// TIA Portal V20 program export: 1 tag tables, 32 data types, 19 data blocks, 60 code blocks (in call order from the OBs), 16 instance data blocks

VAR_GLOBAL   // PLC tag table "IMC88"
   IMC88Sensor_1 AT %I727.0 : Bool;   // High = Sensor active (input type and polarity can be configured)
   IMC88Sensor_2 AT %I727.1 : Bool;   // High = Sensor active (input type and polarity can be configured)
   IMC88Sensor_3 AT %I727.2 : Bool;   // High = Sensor active (input type and polarity can be configured)
   IMC88Sensor_4 AT %I727.3 : Bool;   // High = Sensor active (input type and polarity can be configured)
   IMC88Sensor_5 AT %I727.4 : Bool;
   IMC88Sensor_6 AT %I727.5 : Bool;
   IMC88Sensor_7 AT %I727.6 : Bool;
   IMC88Sensor_8 AT %I727.7 : Bool;
   IMC88IO1 AT %I728.0 : Bool;   // Digital I/O PLC Input PLC Output
   IMC88IO2 AT %I728.1 : Bool;   // Digital I/O PLC Input PLC Output
   IMC88IO3 AT %I728.2 : Bool;   // Digital I/O PLC Input PLC Output
   IMC88IO4 AT %I728.3 : Bool;   // Digital I/O PLC Input PLC Output
   IMC88IO5 AT %I728.4 : Bool;
   IMC88IO6 AT %I728.5 : Bool;
   IMC88IO7 AT %I728.6 : Bool;
   IMC88IO8 AT %I728.7 : Bool;
   "IMC88MotorStateErrorRD -G1.7.4" AT %I729.0 : Bool;   // High = Motor Error; Low = Motor OK
   "IMC88MotorStateErrorRD -G1.7.3" AT %I729.1 : Bool;   // High = Motor Error; Low = Motor OK
   "IMC88MotorStateErrorRD -G1.7.2" AT %I729.2 : Bool;   // High = Motor Error; Low = Motor OK
   "IMC88MotorStateErrorRD -4" AT %I729.3 : Bool;   // High = Motor Error; Low = Motor OK
   "IMC88MotorStateSpeedRD -G1.7.4" AT %IB730 : SInt;   // Speed 0–100 ( 0 = Stop, 100 = max speed), negative sign reverses the turning direction
   "IMC88MotorStateSpeedRD -G1.7.3" AT %IB731 : SInt;   // Speed 0–100 ( 0 = Stop, 100 = max speed), negative sign reverses the turning direction
   "IMC88MotorStateSpeedRD -G1.7.2" AT %IB732 : SInt;   // Speed 0–100 ( 0 = Stop, 100 = max speed), negative sign reverses the turning direction
   "IMC88MotorStateSpeedRD -4" AT %IB733 : SInt;   // Speed 0–100 ( 0 = Stop, 100 = max speed), negative sign reverses the turning direction
   "IMC88MotorCurrentRD -G1.7.4" AT %IW735 : Int;   // Average current in mA
   "IMC88MotorCurrentRD -G1.7.3" AT %IW737 : Int;   // Average current in mA
   "IMC88MotorCurrentRD -G1.7.2" AT %IW739 : Int;   // Average current in mA
   "IMC88MotorCurrentRD -4" AT %IW741 : Int;   // Average current in mA
   "IMC88Voltage(MotorPower)" AT %IW743 : Int;   // Voltage „Motor Power“ in mV
   "IMC88Voltage(Sensors)" AT %IW745 : Int;   // Voltage „Power Logic + Sensors“ in mV
   IMC88Temperature AT %IW747 : Int;   // Temperature in 0,1 C
   IMC88SystemUpTime AT %ID749 : DInt;   // Operating time in seconds since the last start/restart
   "IMC88DigitalOutputRD -G1.7.4" AT %Q535.0 : Bool;
   "IMC88DigitalOutputRD -G1.7.3" AT %Q535.1 : Bool;
   "IMC88DigitalOutputRD -G1.7.2" AT %Q535.2 : Bool;
   "IMC88DigitalOutputRD -4" AT %Q535.3 : Bool;
   "IMC88MotorTargetSpeedRD -G1.7.4" AT %QB536 : SInt;   // Speed 0–100 ( 0 = Stop, 100 = max speed), negative sign reverses the turning direction
   "IMC88MotorTargetSpeedRD -G1.7.3" AT %QB537 : SInt;   // Speed 0–100 ( 0 = Stop, 100 = max speed), negative sign reverses the turning direction
   "IMC88MotorTargetSpeedRD -G1.7.2" AT %QB538 : SInt;   // Speed 0–100 ( 0 = Stop, 100 = max speed), negative sign reverses the turning direction
   "IMC88MotorTargetSpeedRD -4" AT %QB539 : SInt;   // Speed 0–100 ( 0 = Stop, 100 = max speed), negative sign reverses the turning direction
END_VAR

TYPE "BarCode"
// stored: Access Published, Namespace Global
   STRUCT
      "Result Data" : Array[0..63] of Byte;
   END_STRUCT;
END_TYPE

TYPE "ConveyorParameters"
// stored: Access Published, Namespace Global
   STRUCT
      StartUpTime : Time := T#0S;
      SensorFilterTime : Array[1..2] of Time;
      SensorBlockageTime : Time := T#5S;
      EnergySaveTime : Time := T#3s;
      ConvOccTime : Time := T#1000ms;
      "IMC-SpeedSetPoint" : SInt := 100;
   END_STRUCT;
   // SensorFilterTime[1..2] := T#10ms;
END_TYPE

TYPE "ConveyorParameters_TransferUnit"
// stored: Access Published, Namespace Global
   STRUCT
      StartUpTime : Time := T#0S;
      SensorFilterTime : Array[1..2] of Time;
      FrontSensorFilterTime : Array[1..2] of Time;
      "Left/RightSensorFilterTime" : Array[1..2] of Time;
      EndsensorFilterTime : Array[1..2] of Time;
      SensorBlockageTime : Time := T#5S;
      EnergySaveTime : Time := T#3s;
      ConvOccTime : Time := T#1000ms;
   END_STRUCT;
   // SensorFilterTime[1..2] := T#10ms;
   // FrontSensorFilterTime[1..2] := T#10ms;
   // "Left/RightSensorFilterTime"[1..2] := T#10ms;
END_TYPE

TYPE "ConveyorStatus"
// stored: Access Published, Namespace Global
   STRUCT
      Blockage : Bool;
      xReserved_2 : Bool;
      xReserved_3 : Bool;
      xReserved_4 : Bool;
      xReserved_5 : Bool;
      xReserved_6 : Bool;
      xReserved_7 : Bool;
      xReserved_8 : Bool;
      ON : Bool;
      ReadytoRun : Bool;
      Occupied : Bool;
      Running : Bool;
      Fault : Bool;
      Estop : Bool;
      Manual : Bool;
      Stop : Bool;
   END_STRUCT;
END_TYPE

TYPE "EsopZone"
// stored: Access Published, Namespace Global
   STRUCT
      "1" : Bool;
      "2" : Bool;
   END_STRUCT;
END_TYPE

TYPE "Fault"
// stored: Access Published, Namespace Global
   STRUCT
      Motor_Error : Bool;
      Sensor_Blockage : Bool;
   END_STRUCT;
END_TYPE

TYPE "GetDiag"
// stored: Access Published, Namespace Global
   STRUCT
      DiagMode : UInt := 1;
      CommID : HW_ANY;
      ReturnValue : Int;
      CountDiagDetail : UInt;
      MyDiag : DIS;
   END_STRUCT;
END_TYPE

TYPE "ItemDir"
// stored: Access Published, Namespace Global
   STRUCT
      Straight : Bool;
      toRight : Bool;
      toLeft : Bool;
   END_STRUCT;
END_TYPE

TYPE "MABS_Parameters"
// stored: Access Published, Namespace Global
   STRUCT
      StartUpTime : Time := T#5S;
      CrossSensorFilterTime : Array[1..2] of Time;
      SensorBlockageTime : Time := T#5S;
      EnergySaveTime : Time := T#4s;
   END_STRUCT;
END_TYPE

TYPE "ManualInputs"
// stored: Access Published, Namespace Global
   STRUCT
      ManualEnable : Bool;
      Run : Struct
         Forward : Bool;
         Reverse : Bool;
      END_STRUCT;
   END_STRUCT;
END_TYPE

TYPE "S300ForceMode"
// stored: Access Published, Namespace Global
   STRUCT
      BeltDir : Bool;
      RollerDir : Bool;
   END_STRUCT;
END_TYPE

TYPE "S300Manual"
// stored: Namespace Global
   STRUCT
      GoUp : Bool;
      GoStraight : Bool;
      GoLeft : Bool;
      GoRight : Bool;
   END_STRUCT;
END_TYPE

TYPE "SystemSSR"
// stored: Access Published, Namespace Global
   STRUCT
      StartSystem : Bool;   // Start the system
      StopSystem : Bool;   // Stop the system
      ResetSystem : Bool;   // Reset the system
   END_STRUCT;
END_TYPE

TYPE "TrackingData"
// stored: Access Published, Namespace Global
   STRUCT
      Barcode : String;
      ResponseCode : UInt;
      HeightLimit : Bool;
      ActualWeight : Struct
         inRealValue : Real;
         inStringFormat : String;
      END_STRUCT;
      EXIT_1_ : Array[1..1] of Bool;
      EXIT_2_ : Array[1..6] of Bool;
      ToteDir : "Global.ItemDir";
   END_STRUCT;
END_TYPE

TYPE "IB_P01_02_03_in_64bytes_struct"
// stored: Access Published, Namespace Global
   STRUCT
      Reserved : Byte;
      Sens_A : Bool;
      Sens_B : Bool;
      Sens_A_alrm : Bool;
      Sens_B_alrm : Bool;
      Motor_state_A : Bool;
      Motor_state_B : Bool;
      Reserved_1 : Bool;
      Reserved_2 : Bool;
      Fuse_err_A : Bool;
      Back_EMF_err_A : Bool;
      Thermal_err_mot_A : Bool;
      Thermal_err_ctrl_A : Bool;
      Lock_err_A : Bool;
      Unconnected_err_A : Bool;
      Reserved_3 : Bool;
      Reserved_4 : Bool;
      Fuse_err_B : Bool;
      Back_EMF_err_B : Bool;
      Thermal_err_mot_B : Bool;
      Thermal_err_ctrl_B : Bool;
      Lock_err_B : Bool;
      Unconnected_err_B : Bool;
      Reserved_5 : Bool;
      Reserved_6 : Bool;
      Digital_in_1 : Bool;   // NA for IB-P03
      Digital_in_2 : Bool;   // NA for IB-P03
      Digital_in_3 : Bool;   // NA for IB-P03
      Digital_in_4 : Bool;   // NA for IB-P03
      Reserved_7 : Bool;
      Reserved_8 : Bool;
      Reserved_9 : Bool;
      Reserved_10 : Bool;
      Register_Low_D0 : Byte;
      Register_High_D0 : Byte;
      Register_Low_D1 : Byte;
      Register_High_D1 : Byte;
      Register_Low_D2 : Byte;
      Register_High_D2 : Byte;
      Register_Low_D3 : Byte;
      Register_High_D3 : Byte;
      Register_Low_D4 : Byte;
      Register_High_D4 : Byte;
      Register_Low_D5 : Byte;
      Register_High_D5 : Byte;
      Register_Low_D6 : Byte;
      Register_High_D6 : Byte;
      Register_Low_D7 : Byte;
      Register_High_D7 : Byte;
      Register_Low_D8 : Byte;
      Register_High_D8 : Byte;
      Register_Low_D9 : Byte;
      Register_High_D9 : Byte;
      Register_Low_D10 : Byte;
      Register_High_D10 : Byte;
      Register_Low_D11 : Byte;
      Register_High_D11 : Byte;
      Register_Low_D12 : Byte;
      Register_High_D12 : Byte;
      Register_Low_D13 : Byte;
      Register_High_D13 : Byte;
      Register_Low_D14 : Byte;
      Register_High_D14 : Byte;
      Register_Low_D15 : Byte;
      Register_High_D15 : Byte;
      Life_time_mot_A_LL : Byte;
      Life_time_mot_A_LH : Byte;
      Life_time_mot_A_HL : Byte;
      Life_time_mot_A_HH : Byte;
      Life_time_mot_B_LL : Byte;
      Life_time_mot_B_LH : Byte;
      Life_time_mot_B_HL : Byte;
      Life_time_mot_B_HH : Byte;
      Current_mot_A : Byte;
      Current_mot_B : Byte;
      Voltage_mot_A : Byte;
      Voltage_mot_B : Byte;
      Reserved_11 : Array[0..13] of Byte;
   END_STRUCT;
END_TYPE

TYPE "IB_P01_02_03_out_64bytes_struct"
// stored: Access Published, Namespace Global
   STRUCT
      Run_mot_A : Bool;
      Run_mot_B : Bool;
      Reserved_1 : Bool;
      Reserved_2 : Bool;
      Reserved_3 : Bool;
      Reserved_4 : Bool;
      Reserved_5 : Bool;
      Reserved_6 : Bool;
      Speed_1_A : Bool;
      Speed_2_A : Bool;
      Speed_3_A : Bool;
      Speed_4_A : Bool;
      Speed_1_B : Bool;
      Speed_2_B : Bool;
      Speed_3_B : Bool;
      Speed_4_B : Bool;
      Acc_A : Bool;
      Dec_A : Bool;
      Acc_B : Bool;
      Dec_B : Bool;
      Dir_A : Bool;
      Dir_B : Bool;
      Ack_err_A : Bool;
      Ack_err_B : Bool;
      Digital_out1 : Bool;   // NA for IB-P03
      Digital_out2 : Bool;   // NA for IB-P03
      Digital_out3 : Bool;   // NA for IB-P03
      Digital_out4 : Bool;   // NA for IB-P03
      Reserved_7 : Bool;
      Reserved_8 : Bool;
      Reserved_9 : Bool;
      Reserved_10 : Bool;
      Register_Low_D800 : Byte;
      Register_High_D800 : Byte;
      Register_Low_D801 : Byte;
      Register_High_D801 : Byte;
      Register_Low_D802 : Byte;
      Register_High_D802 : Byte;
      Register_Low_D803 : Byte;
      Register_High_D803 : Byte;
      Register_Low_D804 : Byte;
      Register_High_D804 : Byte;
      Register_Low_D805 : Byte;
      Register_High_D805 : Byte;
      Register_Low_D806 : Byte;
      Register_High_D806 : Byte;
      Register_Low_D807 : Byte;
      Register_High_D807 : Byte;
      Register_Low_D808 : Byte;
      Register_High_D808 : Byte;
      Register_Low_D809 : Byte;
      Register_High_D809 : Byte;
      Register_Low_D810 : Byte;
      Register_High_D810 : Byte;
      Register_Low_D811 : Byte;
      Register_High_D811 : Byte;
      Register_Low_D812 : Byte;
      Register_High_D812 : Byte;
      Register_Low_D813 : Byte;
      Register_High_D813 : Byte;
      Register_Low_D814 : Byte;
      Register_High_D814 : Byte;
      Register_Low_D815 : Byte;
      Register_High_D815 : Byte;
      Output_stop : Byte;
      Led_JAM_A : Bool;
      Led_JAM_B : Bool;
      Led_soft1_A : Bool;
      Led_soft1_B : Bool;
      Led_soft2_A : Bool;
      Led_soft2_B : Bool;
      Reserved_11 : Bool;
      Reserved_12 : Bool;
      Reserved_13 : Array[0..25] of Byte;
   END_STRUCT;
END_TYPE

TYPE "MABS"
// stored: Access Published, Namespace Global
   STRUCT
      Run_balls : Bool := false;   // Run transport balls
      Dir_balls : Bool := false;   // 0=forward; 1=backward
      Speed_balls : Int := 90;   // Based on preset speed setting. 60/70/80/90 m/min.
      Switch_left_angle : Int := 45;   // Angle for left transportation 30/180°
      Switch_right_angle : Int := 45;   // Angle for right transportation 30/180°
      Switch_left_to_st_offset : Int := 0;   // Offset angle for straight position from left -8/+10°
      Switch_right_to_st_offset : Int := 0;   // Offset angle for straight position from right -8/+10°
      Init_offset : Int := 0;   // Offset angle for initial position -8/+10°
      Switch_left : Bool := false;   // Swing to left transport direction
      Switch_right : Bool := false;   // Swing to right transport direction
      Switch_left_to_st : Bool := false;   // Swing to straight transport direction CW
      Switch_right_to_st : Bool := false;   // Swing to straight transport direction CCW
      EMS : Bool := false;   // Inhib controls and reset MABS initialisation
      Init : Bool := false;   // Run MABS initialisation sequence (if not done)
      Init_done : Bool := false;   // MABS initialisation sequence done
      Ready : Bool := false;   // MABS no error, initialisation done, communication OK
      Init_sensor : Bool := false;   // MABS straight position sensor
      Left_Pos_reach : Bool := false;   // MABS transport balls in left position
      Right_Pos_reach : Bool := false;   // MABS transport balls in right position
      Straight_Pos_reach : Bool := false;   // MABS transport balls in straight position
      Error_motA : Bool := false;   // Hardware error motor A
      Error_motB : Bool := false;   // Hardware error motor B
      Error_timeout_sw : Bool := false;   // Swing motor timeout
      Error_com : Bool := false;   // Communication error (life bit, 5s delayed)
      Error : Bool := false;   // Error synthesis
      Reset_error : Bool := false;   // Reset all errors
      Timeout_val : Time := T#10s;   // Swing timeout value
      HMI_sts : UInt := 0;   // Sts word for HMI (0=Off; 1=Running; 2=Init requested; 4=Error )
   END_STRUCT;
END_TYPE

TYPE "MABS_ManIn"
// stored: Access Published, Namespace Global
   STRUCT
      RunBalls : Bool;
      Switch : Struct
         ToLeft : Bool;
         ToRight : Bool;
         left_to_st : Bool;
         right_to_st : Bool;
      END_STRUCT;
   END_STRUCT;
END_TYPE

TYPE "MABS_Setpoint"
// stored: Access Published, Namespace Global
   STRUCT
      ChangeBallsDirection : Bool;   // 0=forward; 1=backward
      Speed_balls : Int := 0;   // Based on preset speed setting. 60/70/80/90 m/min.
      Init_offset : Int;   // Offset angle for initial position -8/+10°
   END_STRUCT;
END_TYPE

TYPE "Log_Data_Byte_Decimal"
// stored: Namespace ProductionLine
   STRUCT
      DataType : Int;
      Representation : Int;
      RepreLength : Int;
      Reserve : Int;
      Data : Int;
   END_STRUCT;
END_TYPE

TYPE "Log_Data_Char"
// stored: Namespace ProductionLine
   STRUCT
      DataType : Byte;
      Representation : Byte;
      RepreLength : Byte;
      Reserve : Byte;
      Data : Char;
   END_STRUCT;
END_TYPE

TYPE "Log_Data_String20"
// stored: Namespace ProductionLine
   STRUCT
      DataType : Byte;
      Representation : Byte;
      RepreLength : Byte;
      Reserve : Byte;
      Data : String[20];
   END_STRUCT;
END_TYPE

TYPE "Log_LogMsg_Header"
// stored: Namespace ProductionLine
   STRUCT
      STX : Byte;
      SOH : Byte;
      MsgLength : Int;
      MsgType : Byte;
      Reserve : Byte;
      EventLevel : Byte;
      EventGroup : Byte;
      Timestamp : Date_And_Time;
      EventID : Int;
   END_STRUCT;
END_TYPE

TYPE "OPC_DestAssign"
// stored: Namespace ProductionLine
   STRUCT
      SourceSeq : Int;
      SourceNode : String[8];
      TotesID : String[10];
      WMSID : String[20];
      DestinationNode : String[8];
   END_STRUCT;
END_TYPE

TYPE "OPC_DestAssign_Ack"
// stored: Namespace ProductionLine
   STRUCT
      AckSeq : Int;
      SourceNode : String[8];
      TotesID : String[10];
      WMSID : String[20];
      Confirmation : String[1];
   END_STRUCT;
END_TYPE

TYPE "OPC_DestInfo"
// stored: Namespace ProductionLine
   STRUCT
      SourceSeq : Int;   // //Communication flag, described in the Request - Response tab
      DecisionPoint : String[30];   // // Machine/workstation code: - DP1,…, DP4
      Barcode : String[30];   // // Unique identification of scanned KLTs. For NoRead use ??????????
      InformationPoint : String[30];   // // Identification of the target location: - IP1...IP9
   END_STRUCT;
END_TYPE

TYPE "OPC_DestInfo_Ack"
// stored: Namespace ProductionLine
   STRUCT
      AckSeq : Int;   // //Communication flag, described in the Data tab
   END_STRUCT;
END_TYPE

TYPE "OPC_DestRequest_Ack"
// stored: Namespace ProductionLine
   STRUCT
      AckSeq : Int;   // //Communication flag, described in the Request - Response tab
      DecisionPoint : String[30];   // // Machine/workstation code:- DP1,…, DP4
      Barcode : String[30];   // // Unique identification of scanned KLTs. For NoRead use ??????????
      State : String[10];   // // Response status: - OK = task ready - NG (not good) = error
      Destination : String[30];   // Identification of the target location: - IP1...IP9
      ErrorReason : String[150];   // // Reason for error in case of status = NG.
   END_STRUCT;
END_TYPE

TYPE "OPC_DsetRequest"
// stored: Namespace ProductionLine
   STRUCT
      SourceSeq : Int;   // // Communication flag, described in the Request - Response tab
      DecisionPoint : String[30];   // // Machine/workstation code: - DP1,…, DP4
      Barcode : String[30];   // // Unique identification of scanned KLTs. For NoRead use ??????????
   END_STRUCT;
END_TYPE

TYPE "OPC_SegmentStatus"
// stored: Namespace ProductionLine
   STRUCT
      Segment : Struct
         FlowRackLoop : Int;
         FlowRackWorkplaceLeft : Int;
         FlowRackWorkplaceRight : Int;
         FragileLoop : Int;
      END_STRUCT;
   END_STRUCT;
END_TYPE

TYPE "OPC_SystStatus_Ack"
// stored: Namespace ProductionLine
   STRUCT
      AckSeq : Int;
   END_STRUCT;
END_TYPE

TYPE "OPC_SystemStatus"
// stored: Namespace ProductionLine
   STRUCT
      SourceSeq : Int;
   END_STRUCT;
END_TYPE

DATA_BLOCK "DB_Sync"   // DB3
{ S7_Optimized_Access := 'TRUE' }
// stored: MemoryReserve 100
   VAR
      memoryBit : Struct
         System_Byte : Byte;
         FirstScan : Bool;
         DiagStatusUpdate : Bool;
         AlwaysTRUE : Bool;
         AlwaysFALSE : Bool;
      END_STRUCT;
      ClockBit : Struct
         Clock_Byte : Byte;
         Clock_10Hz : Bool;
         Clock_5Hz : Bool;
         "Clock_2.5Hz" : Bool;
         Clock_2Hz : Bool;
         "Clock_1.25Hz" : Bool;
         Clock_1Hz : Bool;
         "Clock_0.625Hz" : Bool;
         "Clock_0.5Hz" : Bool;
      END_STRUCT;
      startbit1 : Bool;
      stopbit1 : Bool;
      resetbit1 : Bool;
      startbit2 : Bool;
      stopbit2 : Bool;
      resetbit2 : Bool;
   END_VAR
BEGIN
END_DATA_BLOCK

DATA_BLOCK "DB_SafetyStandard"   // DB20
// stored: Access Published, MemoryReserve 100
   VAR
      ToStandard : Struct
         EstopActive : Bool;
      END_STRUCT;
      PressReset : Bool;
      ToHMI : Struct
         "EstopPB -MCC001+MCC001-SF1" : Bool;
         "EstopPB -ZONA1+A1.1.1-SF1" : Bool;
         "EstopPB -ZONA1+A1.1.10-SF1" : Bool;
         "EstopPB -ZONA1+A1.2.1-SF1" : Bool;
         "EstopPB -ZONA1+B1.22.1-SF1" : Bool;
         "EstopPB -ZONA1+C1.3.1-SF1" : Bool;
         "EstopPB -ZONA1+B1.12.1-SF1" : Bool;
         "EstopPB -ZONA1+B1.15.1-SF1" : Bool;
         "EstopPB -ZONA1+B1.17.3-SF1" : Bool;
         "EstopPB -ZONA2+D1.11.1-SF1" : Bool;
         "EstopPB -ZONA2+E1.1.2-SF1" : Bool;
         "EstopPB -ZONA2+A1.10.3-SF1" : Bool;
         "EstopPB -ZONA2+A1.12.1-SF1" : Bool;
         "EstopPB -ZONA2+A1.16.8-SF1" : Bool;
         "EstopPB -ZONA2+B1.17.0-SF1" : Bool;
         "EstopPB -ZONA2+A2.4.5-SF1" : Bool;
         "EstopPB -ZONA2+G1.5.3-SF1" : Bool;
         "EstopPB -ZONA2+G1.7.1-SF1" : Bool;
         "PhaseOK -MCC001" : Bool;
      END_STRUCT;
      holdAlarmOffTimer : TON_TIME;
      holdAlarmOff : Bool;
   END_VAR
BEGIN
END_DATA_BLOCK

DATA_BLOCK "DB_Temporary"   // DB40
// stored: MemoryReserve 100, Namespace EmptyLine
   VAR
      MABS1_In { ExternalAccessible := 'False'; ExternalVisible := 'False'; ExternalWritable := 'False'} : "Global.IB_P01_02_03_in_64bytes_struct";
      MABS1_Out { ExternalAccessible := 'False'; ExternalVisible := 'False'; ExternalWritable := 'False'} : "Global.IB_P01_02_03_out_64bytes_struct";
      MABS2_In { ExternalAccessible := 'False'; ExternalVisible := 'False'; ExternalWritable := 'False'} : "Global.IB_P01_02_03_in_64bytes_struct";
      MABS2_Out { ExternalAccessible := 'False'; ExternalVisible := 'False'; ExternalWritable := 'False'} : "Global.IB_P01_02_03_out_64bytes_struct";
   END_VAR
BEGIN
END_DATA_BLOCK

DATA_BLOCK "ToteDir"   // DB43
// stored: MemoryReserve 100, Namespace EmptyLine
   VAR
      Conveyor : Array[_."J1.6.1".._."J1.6.2"] of "Global.ItemDir";
   END_VAR
BEGIN
END_DATA_BLOCK

DATA_BLOCK "DB_Global"   // DB23
// stored: Access Published, MemoryReserve 100, Namespace Global
   VAR
      Status : Struct
         Line : Struct
            ProductionLine : Struct
               On : Array[_.gminProductionLine.._.gmaxProductionLine] of Bool;
               ReadyToRun : Array[_.gminProductionLine.._.gmaxProductionLine] of Bool;
               Occupied : Array[_.gminProductionLine.._.gmaxProductionLine] of Bool;
               Running : Array[_.gminProductionLine.._.gmaxProductionLine] of Bool;
               Fault : Array[_.gminProductionLine.._.gmaxProductionLine] of Bool;
               Estop : Array[_.gminProductionLine.._.gmaxProductionLine] of Bool;
               Manual : Array[_.gminProductionLine.._.gmaxProductionLine] of Bool;
               Stop : Array[_.gminProductionLine.._.gmaxProductionLine] of Bool;
               Blockage : Array[_.gminProductionLine.._.gmaxProductionLine] of Bool;
            END_STRUCT;
            EmptyLine : Struct
               On : Array[_.gminEmptyLine.._.gmaxEmptyLine] of Bool;
               ReadyToRun : Array[_.gminEmptyLine.._.gmaxEmptyLine] of Bool;
               Occupied : Array[_.gminEmptyLine.._.gmaxEmptyLine] of Bool;
               Running : Array[_.gminEmptyLine.._.gmaxEmptyLine] of Bool;
               Fault : Array[_.gminEmptyLine.._.gmaxEmptyLine] of Bool;
               Estop : Array[_.gminEmptyLine.._.gmaxEmptyLine] of Bool;
               Manual : Array[_.gminEmptyLine.._.gmaxEmptyLine] of Bool;
               Stop : Array[_.gminEmptyLine.._.gmaxEmptyLine] of Bool;
               Blockage : Array[_.gminEmptyLine.._.gmaxEmptyLine] of Bool;
            END_STRUCT;
            PackedLine : Struct
               On : Array[_.gminPackedLine.._.gmaxPackedLine] of Bool;
               ReadyToRun : Array[_.gminPackedLine.._.gmaxPackedLine] of Bool;
               Occupied : Array[_.gminPackedLine.._.gmaxPackedLine] of Bool;
               Running : Array[_.gminPackedLine.._.gmaxPackedLine] of Bool;
               Fault : Array[_.gminPackedLine.._.gmaxPackedLine] of Bool;
               Estop : Array[_.gminPackedLine.._.gmaxPackedLine] of Bool;
               Manual : Array[_.gminPackedLine.._.gmaxPackedLine] of Bool;
               Stop : Array[_.gminPackedLine.._.gmaxPackedLine] of Bool;
               Blockage : Array[_.gminPackedLine.._.gmaxPackedLine] of Bool;
            END_STRUCT;
         END_STRUCT;
      END_STRUCT;
   END_VAR
BEGIN
   // Status.Line.ProductionLine.On[1001] : AS1.1.1
   // Status.Line.ProductionLine.On[1002] : AS1.1.2
   // Status.Line.ProductionLine.ReadyToRun[1001] : AS1.1.1
   // Status.Line.ProductionLine.ReadyToRun[1002] : AS1.1.2
   // Status.Line.ProductionLine.Occupied[1001] : AS1.1.1
   // Status.Line.ProductionLine.Occupied[1002] : AS1.1.2
   // Status.Line.ProductionLine.Running[1001] : AS1.1.1
   // Status.Line.ProductionLine.Running[1002] : AS1.1.2
   Status.Line.ProductionLine.Fault[1001] := 0;   // AS1.1.1
   Status.Line.ProductionLine.Fault[1002] := 0;   // AS1.1.2
   Status.Line.ProductionLine.Estop[1001] := 0;   // AS1.1.1
   Status.Line.ProductionLine.Estop[1002] := 0;   // AS1.1.2
   Status.Line.ProductionLine.Manual[1001] := 0;   // AS1.1.1
   Status.Line.ProductionLine.Manual[1002] := 0;   // AS1.1.2
   Status.Line.ProductionLine.Stop[1001] := 0;   // AS1.1.1
   Status.Line.ProductionLine.Stop[1002] := 0;   // AS1.1.2
   Status.Line.ProductionLine.Blockage[1001] := 0;   // AS1.1.1
   Status.Line.ProductionLine.Blockage[1002] := 0;   // AS1.1.2
   // Status.Line.PackedLine.ReadyToRun[3001] : BP1.1.1
   // Status.Line.PackedLine.ReadyToRun[3002] : BP1.1.2
   // Status.Line.PackedLine.Occupied[3001] : BP1.1.1
   // Status.Line.PackedLine.Occupied[3002] : BP1.1.2
   // Status.Line.PackedLine.Running[3001] : BP1.1.1
   // Status.Line.PackedLine.Running[3002] : BP1.1.2
   // Status.Line.PackedLine.Fault[3001] : BP1.1.1
   // Status.Line.PackedLine.Fault[3002] : BP1.1.2
   // Status.Line.PackedLine.Estop[3001] : BP1.1.1
   // Status.Line.PackedLine.Estop[3002] : BP1.1.2
   // Status.Line.PackedLine.Manual[3001] : BP1.1.1
   // Status.Line.PackedLine.Manual[3002] : BP1.1.2
   // Status.Line.PackedLine.Stop[3001] : BP1.1.1
   // Status.Line.PackedLine.Stop[3002] : BP1.1.2
   // Status.Line.PackedLine.Blockage[3001] : BP1.1.1
   // Status.Line.PackedLine.Blockage[3002] : BP1.1.2
END_DATA_BLOCK

DATA_BLOCK "DB_ConveyorParameters"   // DB26
// stored: Access Published, MemoryReserve 100, Namespace EmptyLine
   VAR
      Line : Struct
         EmptyLine : Struct
            Conveyor : Array[_.minEmptyLine.._.maxEmptyLine] of "Global.ConveyorParameters";
            Mabs { S7_SetPoint := 'True'} : Array[_."J1.6.1".._."J1.6.2"] of "Global.MABS_Parameters";
         END_STRUCT;
      END_STRUCT;
   END_VAR
BEGIN
END_DATA_BLOCK

DATA_BLOCK "DB_Manual"   // DB18
// stored: Access Published, MemoryReserve 100, Namespace EmptyLine
   VAR
      Conveyor : Struct
         ID : Int;
         Enable : Bool;
         Run : Bool;
         in : Bool;
      END_STRUCT;
      Line : Struct
         EmptyLine : Struct
            Conveyor { S7_SetPoint := 'True'} : Array[_.minEmptyLine.._.maxEmptyLine] of "Global.ManualInputs";
         END_STRUCT;
      END_STRUCT;
   END_VAR
BEGIN
END_DATA_BLOCK

DATA_BLOCK "DB_UDI"   // DB37
// stored: MemoryReserve 100, Namespace EmptyLine
   VAR
      EmptyLine : Struct
         Upstream : Struct
            Conveyor : Array[_.minEmptyLine.._.maxEmptyLine] of Bool;
         END_STRUCT;
         DownstreamAcu : Struct
            Stop : Struct
               Conveyor : Array[_.minEmptyLine.._.maxEmptyLine] of Bool;
            END_STRUCT;
         END_STRUCT;
         Interlock : Struct
            Stop : Struct
               Conveyor : Array[_.minEmptyLine.._.maxEmptyLine] of Bool;
            END_STRUCT;
         END_STRUCT;
         Fault : Struct
            Stop : Struct
               Conveyor : Array[_.minEmptyLine.._.maxEmptyLine] of Bool;
            END_STRUCT;
         END_STRUCT;
         Transfer : Struct
            "B1.6.1" : Struct
               "Upstream Straight" : Bool;
               "Upstream Arm" : Bool;
            END_STRUCT;
         END_STRUCT;
      END_STRUCT;
   END_VAR
BEGIN
END_DATA_BLOCK

DATA_BLOCK "DB_Alarm"   // DB14
// stored: Access Published, MemoryReserve 100, Namespace EmptyLine
   VAR
      "word" : Struct
         Line : Struct
            EmptyLine : Struct
               Conveyor : Array[_.minEmptyLine.._.maxEmptyLine] of Word;
            END_STRUCT;
         END_STRUCT;
      END_STRUCT;
      Simu : Word;
   END_VAR
BEGIN
END_DATA_BLOCK

DATA_BLOCK "DB_SystemSSR"   // DB5
// stored: Access Published, MemoryReserve 100, Namespace Global
   VAR
      FromHMI : Struct
         Line : Struct
            ProductionLine : "Global.SystemSSR";
            EmptyLine { S7_SetPoint := 'True'} : "Global.SystemSSR";
            PackedLine { S7_SetPoint := 'True'} : "Global.SystemSSR";
         END_STRUCT;
      END_STRUCT;
      Line : Struct
         ProductionLine : "Global.SystemSSR";
         EmptyLine { S7_SetPoint := 'True'} : "Global.SystemSSR";
         PackedLine { S7_SetPoint := 'True'} : "Global.SystemSSR";
      END_STRUCT;
      Zone : Struct
         "1" : "Global.SystemSSR";
         "2" : "Global.SystemSSR";
      END_STRUCT;
   END_VAR
BEGIN
END_DATA_BLOCK

DATA_BLOCK "DB_SystemSimu"   // DB30
// stored: Access Published, MemoryReserve 100, Namespace Global
   VAR
      TriggerSensor : Struct
         Line : Struct
            ProductionLine : Struct
               Conveyor : Array[_.gminProductionLine.._.gmaxProductionLine] of Bool;
            END_STRUCT;
            EmptyLine : Struct
               Conveyor : Array[_.gminEmptyLine.._.gmaxEmptyLine] of Bool;
            END_STRUCT;
            PackedLine : Struct
               Conveyor : Array[_.gminPackedLine.._.gmaxPackedLine] of Bool;
            END_STRUCT;
         END_STRUCT;
      END_STRUCT;
      TriggerFault : Struct
         Line : Struct
            ProductionLine : Struct
               Conveyor : Array[_.gminProductionLine.._.gmaxProductionLine] of Bool;
            END_STRUCT;
            EmptyLine : Struct
               Conveyor : Array[_.gminEmptyLine.._.gmaxEmptyLine] of Bool;
            END_STRUCT;
            PackedLine : Struct
               Conveyor : Array[_.gminPackedLine.._.gmaxPackedLine] of Bool;
            END_STRUCT;
         END_STRUCT;
      END_STRUCT;
      Fire : Bool;
      DatamanResultsAvailable : Bool;
   END_VAR
BEGIN
   // TriggerSensor.Line.ProductionLine.Conveyor[1001] : AS1.1.1
   // TriggerSensor.Line.ProductionLine.Conveyor[1002] : AS1.1.2
   // TriggerFault.Line.ProductionLine.Conveyor[1001] : AS1.1.1
   // TriggerFault.Line.ProductionLine.Conveyor[1002] : AS1.1.2
END_DATA_BLOCK

DATA_BLOCK "DB_VisuColor"   // DB2
// stored: Access Published, MemoryReserve 100, Namespace Global
   VAR
      Line : Struct
         ProductionLine : Struct
            GlobalStatus : Int;
            Conveyor : Array[_.gminProductionLine.._.gmaxProductionLine] of Int;
         END_STRUCT;
         EmptyLine : Struct
            GlobalStatus : Int;
            Conveyor : Array[_.gminEmptyLine.._.gmaxEmptyLine] of Int;
         END_STRUCT;
         PackedLine : Struct
            GlobalStatus : Int;
            Conveyor : Array[_.gminPackedLine.._.gmaxPackedLine] of Int;
         END_STRUCT;
      END_STRUCT;
   END_VAR
BEGIN
END_DATA_BLOCK

DATA_BLOCK "DB_AsiSetpoint"   // DB24
// stored: Access Published, MemoryReserve 100, Namespace EmptyLine
   VAR
      Line : Struct
         EmptyLine : Struct
            DirChange : Struct
               Conveyor : Array[_.minEmptyLine.._.maxEmptyLine] of Bool;
            END_STRUCT;
            Speed : Struct
               Conveyor : Array[_.minEmptyLine.._.maxEmptyLine] of Bool;
            END_STRUCT;
         END_STRUCT;
      END_STRUCT;
   END_VAR
BEGIN
END_DATA_BLOCK

DATA_BLOCK "DB_NordSetPoint"   // DB35
// stored: Access Published, MemoryReserve 100, Namespace EmptyLine
   VAR
      Line : Struct
         EmptyLine : Struct   // -(0 - 16000) -> (CW: 0 - 100%) || +(0 - 16000) (CCW: 0 - 100%) || freq. has been set via NORDCON
            Conveyor : Array[_.minEmptyLine.._.maxEmptyLine] of DInt;
         END_STRUCT;
      END_STRUCT;
   END_VAR
BEGIN
END_DATA_BLOCK

DATA_BLOCK "DB_S300SetPoint"   // DB21
// stored: MemoryReserve 100, Namespace Global
   VAR
      Line : Struct
         ProductionLine : Struct
            DirChange : Struct
               Conveyor : Array[_.gminProductionLine.._.gmaxProductionLine] of "Global.S300ForceMode";
            END_STRUCT;
         END_STRUCT;
      END_STRUCT;
   END_VAR
BEGIN
END_DATA_BLOCK

DATA_BLOCK "Expedtion"   // DB4
// stored: MemoryReserve 100, Namespace ProductionLine
   VAR
      ExpedtionDirection : Int;
      ExpedtionEnable : Bool;
      CurrentExpedtionDirection : String;
      StraightTableselection : Int;
      CurrentStraightTableselection : String;
      LeftTableselection : Int;
      CurrentLeftTableselection : String;
      StraightTableselectionEnable : Bool;
      LeftTableselectionEnable : Bool;
   END_VAR
BEGIN
END_DATA_BLOCK

DATA_BLOCK "DB_LogMsg"   // DB39
// stored: MemoryReserve 100, Namespace ProductionLine
   VAR
      Write_Position : Int;
      abyLogMsg_Buffer : Array[0..8191] of Byte;
      LogMsg_1 : Struct
         Para_BYTE_02 : "ProductionLine.Log_Data_Byte_Decimal";
      END_STRUCT;
      LogMsg_2 : Struct
         Para_BYTE_02 : "ProductionLine.Log_Data_Byte_Decimal";
      END_STRUCT;
      LogMsg_3 : Struct
         Para_BYTE_02 : "ProductionLine.Log_Data_Byte_Decimal";
      END_STRUCT;
      LogMsg_4 : Struct
         Para_STRING_01 : "ProductionLine.Log_Data_String20";
         Para_BYTE_02 : "ProductionLine.Log_Data_Byte_Decimal";
         Para_STRING_05 : "ProductionLine.Log_Data_String20";
      END_STRUCT;
      LogMsg_5 : Struct
         Para_STRING_01 : "ProductionLine.Log_Data_String20";
         Para_BYTE_02 : "ProductionLine.Log_Data_Byte_Decimal";
         Para_STRING_03 : "ProductionLine.Log_Data_String20";
         Para_STRING_05 : "ProductionLine.Log_Data_String20";
      END_STRUCT;
      LogMsg_6 : Struct
         Para_STRING_01 : "ProductionLine.Log_Data_String20";
         Para_BYTE_02 : "ProductionLine.Log_Data_Byte_Decimal";
      END_STRUCT;
      LogMsg_7 : Struct
         Para_STRING_01 : "ProductionLine.Log_Data_String20";
         Para_BYTE_02 : "ProductionLine.Log_Data_Byte_Decimal";
         Para_STRING_03 : "ProductionLine.Log_Data_String20";
         Para_STRING_04 : "ProductionLine.Log_Data_String20";
      END_STRUCT;
      LogMsg_8 : Struct
         Para_STRING_01 : "ProductionLine.Log_Data_String20";
         Para_BYTE_02 : "ProductionLine.Log_Data_Byte_Decimal";
      END_STRUCT;
      LogMsg_9 : Struct
         Para_STRING_01 : "ProductionLine.Log_Data_String20";
         Para_BYTE_02 : "ProductionLine.Log_Data_Byte_Decimal";
         Para_STRING_03 : "ProductionLine.Log_Data_String20";
         Para_STRING_04 : "ProductionLine.Log_Data_String20";
         Para_STRING_05 : "ProductionLine.Log_Data_String20";
      END_STRUCT;
      LogMsg_10 : Struct
         Para_STRING_01 : "ProductionLine.Log_Data_String20";
         Para_BYTE_02 : "ProductionLine.Log_Data_Byte_Decimal";
         Para_STRING_03 : "ProductionLine.Log_Data_String20";
         Para_STRING_04 : "ProductionLine.Log_Data_String20";
         Para_CHAR_05 : "ProductionLine.Log_Data_Char";
      END_STRUCT;
   END_VAR
BEGIN
END_DATA_BLOCK

DATA_BLOCK "OPC_Data"   // DB41
// stored: MemoryReserve 0, Namespace ProductionLine
   VAR
      Watchdog : Struct
         Keep_Alive_PLC : Int;   // //Periodic counter, incremented every 10 seconds. If one side does not increment the counter within 30 seconds, it will be considered offline by the other side.
         Keep_Alive_WMS : Int;   // //Periodic counter, incremented every 10 seconds. If one side does not increment the counter within 30 seconds, it will be considered offline by the other side.
      END_STRUCT;
      DP1 : Struct
         DestRequest : Struct
            Source : "ProductionLine.OPC_DsetRequest";
            Ack { S7_SetPoint := 'True'} : "ProductionLine.OPC_DestRequest_Ack";
         END_STRUCT;
      END_STRUCT;
      DP2 : Struct
         DestRequest : Struct
            Source : "ProductionLine.OPC_DsetRequest";
            Ack { S7_SetPoint := 'True'} : "ProductionLine.OPC_DestRequest_Ack";
         END_STRUCT;
      END_STRUCT;
      DP3 : Struct
         DestRequest : Struct
            Source : "ProductionLine.OPC_DsetRequest";
            Ack { S7_SetPoint := 'True'} : "ProductionLine.OPC_DestRequest_Ack";
         END_STRUCT;
      END_STRUCT;
      DP4 : Struct
         DestRequest : Struct
            Source : "ProductionLine.OPC_DsetRequest";
            Ack { S7_SetPoint := 'True'} : "ProductionLine.OPC_DestRequest_Ack";
         END_STRUCT;
      END_STRUCT;
      IP1 : Struct
         DestInfo : Struct
            Source : "ProductionLine.OPC_DestInfo";
            Ack { S7_SetPoint := 'True'} : "ProductionLine.OPC_DestInfo_Ack";
         END_STRUCT;
      END_STRUCT;
      IP2 : Struct
         DestInfo : Struct
            Source : "ProductionLine.OPC_DestInfo";
            Ack { S7_SetPoint := 'True'} : "ProductionLine.OPC_DestInfo_Ack";
         END_STRUCT;
      END_STRUCT;
      IP3 : Struct
         DestInfo : Struct
            Source : "ProductionLine.OPC_DestInfo";
            Ack { S7_SetPoint := 'True'} : "ProductionLine.OPC_DestInfo_Ack";
         END_STRUCT;
      END_STRUCT;
      IP4 : Struct
         DestInfo : Struct
            Source : "ProductionLine.OPC_DestInfo";
            Ack { S7_SetPoint := 'True'} : "ProductionLine.OPC_DestInfo_Ack";
         END_STRUCT;
      END_STRUCT;
      IP5 : Struct
         DestInfo : Struct
            Source : "ProductionLine.OPC_DestInfo";
            Ack { S7_SetPoint := 'True'} : "ProductionLine.OPC_DestInfo_Ack";
         END_STRUCT;
      END_STRUCT;
      IP6 : Struct
         DestInfo : Struct
            Source : "ProductionLine.OPC_DestInfo";
            Ack { S7_SetPoint := 'True'} : "ProductionLine.OPC_DestInfo_Ack";
         END_STRUCT;
      END_STRUCT;
      IP7 : Struct
         DestInfo : Struct
            Source : "ProductionLine.OPC_DestInfo";
            Ack { S7_SetPoint := 'True'} : "ProductionLine.OPC_DestInfo_Ack";
         END_STRUCT;
      END_STRUCT;
      IP8 : Struct
         DestInfo : Struct
            Source : "ProductionLine.OPC_DestInfo";
            Ack { S7_SetPoint := 'True'} : "ProductionLine.OPC_DestInfo_Ack";
         END_STRUCT;
      END_STRUCT;
      IP9 : Struct
         DestInfo : Struct
            Source : "ProductionLine.OPC_DestInfo";
            Ack { S7_SetPoint := 'True'} : "ProductionLine.OPC_DestInfo_Ack";
         END_STRUCT;
      END_STRUCT;
      Status : "ProductionLine.OPC_SegmentStatus";
   END_VAR
BEGIN
   DP1.DestRequest.Source.DecisionPoint := 'DP1';
   DP2.DestRequest.Source.DecisionPoint := 'DP2';
   DP3.DestRequest.Source.DecisionPoint := 'DP3';
   DP4.DestRequest.Source.DecisionPoint := 'DP4';
   IP1.DestInfo.Source.DecisionPoint := 'DP1';
   IP2.DestInfo.Source.DecisionPoint := 'DP1';
   IP3.DestInfo.Source.DecisionPoint := 'DP2';
   IP4.DestInfo.Source.DecisionPoint := 'DP2';
   IP5.DestInfo.Source.DecisionPoint := 'DP2';
   IP6.DestInfo.Source.DecisionPoint := 'DP3';
   IP7.DestInfo.Source.DecisionPoint := 'DP3';
   IP8.DestInfo.Source.DecisionPoint := 'DP4';
   IP9.DestInfo.Source.DecisionPoint := 'DP4';
END_DATA_BLOCK

DATA_BLOCK "DB_ToteTracking"   // DB15
// stored: MemoryReserve 100, Namespace ProductionLine
   VAR
      Conveyor : Array[_.minProductionLine.._.maxProductionLine] of "Global.TrackingData";
      Barcode : Array[_.minProductionLine.._.maxProductionLine] of String;
      Transfer : Array[_.minProductionLine.._.maxProductionLine] of "Global.ItemDir";
   END_VAR
BEGIN
END_DATA_BLOCK

ORGANIZATION_BLOCK "Main"   // OB1, LAD, ProgramCycle
TITLE = "Main Program Sweep (Cycle)"
{ S7_Optimized_Access := 'TRUE' }
// stored: SetENOAutomatically false
   VAR_INPUT
      Initial_Call : Bool;   // Initial call of this OB
      Remanence : Bool;   // =True, if remanent data are available
   END_VAR
BEGIN

REGION Network 1
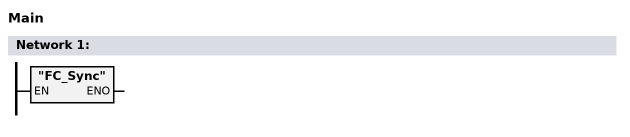
   RUNG wire#powerrail
      "FC_Sync"()
   END_RUNG
   // the same network as SCL:
   "FC_Sync"();
END_REGION
END_ORGANIZATION_BLOCK

FUNCTION "FC_Sync" : Void
{ S7_Optimized_Access := 'TRUE' }
VERSION : 0.1

BEGIN
	
	
	
	REGION system memory bits
	    
	    "DB_Sync".memoryBit.System_Byte := "System_Byte";
	    "DB_Sync".memoryBit.FirstScan := "FirstScan";
	    "DB_Sync".memoryBit.DiagStatusUpdate := "DiagStatusUpdate";
	    "DB_Sync".memoryBit.AlwaysTRUE := "AlwaysTRUE";
	    "DB_Sync".memoryBit.AlwaysFALSE := "AlwaysFALSE";
	    
	END_REGION
	
	REGION clock memory bits
	    
	    "DB_Sync".ClockBit.Clock_Byte := "Clock_Byte";
	    "DB_Sync".ClockBit."Clock_10Hz" := "Clock_10Hz";
	    "DB_Sync".ClockBit."Clock_5Hz" := "Clock_5Hz";
	    "DB_Sync".ClockBit."Clock_2.5Hz" := "Clock_2.5Hz";
	    "DB_Sync".ClockBit."Clock_2Hz" := "Clock_2Hz";
	    "DB_Sync".ClockBit."Clock_1.25Hz" := "Clock_1.25Hz";
	    "DB_Sync".ClockBit."Clock_1Hz" := "Clock_1Hz";
	    "DB_Sync".ClockBit."Clock_0.625Hz" := "Clock_0.625Hz";
	    "DB_Sync".ClockBit."Clock_0.5Hz" := "Clock_0.5Hz";
	    
	END_REGION
	
	
	REGION Start/Stop/Reset 
	    //Zone 1 
	    "DB_Sync".startbit1 := "startBit1";
	    "DB_Sync".stopbit1 := "stopBit1";
	    "DB_Sync".resetbit1 := "ResetBit1";
	    
	    //Zone 2 
	    "DB_Sync".startbit2 := "startBit2";
	    "DB_Sync".stopbit2 := "stopBit2";
	    "DB_Sync".resetbit2 := "ResetBit2";
	END_REGION
	
	
	
	
	
	
	
	
	
	
	
	
	
	
	
	
	
	
END_FUNCTION

FUNCTION_BLOCK "FSFB_Main_Safety_RTG1"   // FB1, F_LAD
   VAR
      AllStopZone1 { ExternalAccessible := 'False'; ExternalVisible := 'False'; ExternalWritable := 'False'} : Bool;
      AllStopZone2 : Bool;
      Reset : Bool;
      Pair1 : ESTOP1;
      Pair2 : ESTOP1;
      Pair3 : ESTOP1;
      Pair4 : ESTOP1;
      Pair5 : ESTOP1;
      Pair6 : ESTOP1;
      Pair7 : ESTOP1;
      Pair8 : ESTOP1;
      Pair9 : ESTOP1;
      Pair10 : ESTOP1;
      ACK_GL : ACK_GL;
      ResetDelayTimer_Pair1 : TOF;
      ResetDelayTimer_Pair2 : TOF;
      ResetDelayTimer_Pair3 : TOF;
      ResetDelayTimer_Pair4 : TOF;
      ResetDelayTimer_Pair5 : TOF;
      ResetDelayTimer_Pair6 : TOF;
      ResetDelayTimer_Pair7 : TOF;
      ResetDelayTimer_Pair8 : TOF;
      ResetDelayTimer_Pair9 : TOF;
      ResetDelayTimer_Pair10 : TOF;
      mem_Pair1 : Bool;
      mem_Pair2 : Bool;
      mem_Pair3 : Bool;
      mem_Pair4 : Bool;
      mem_Pair5 : Bool;
      mem_Pair6 : Bool;
      mem_Pair7 : Bool;
      mem_Pair8 : Bool;
      mem_Pair9 : Bool;
      mem_Pair10 : Bool;
   END_VAR
   VAR_TEMP   // added for the SCL form of the ladder/FBD networks
      _w1 : Bool;
   END_VAR
BEGIN

REGION Network 1
   // Zone1
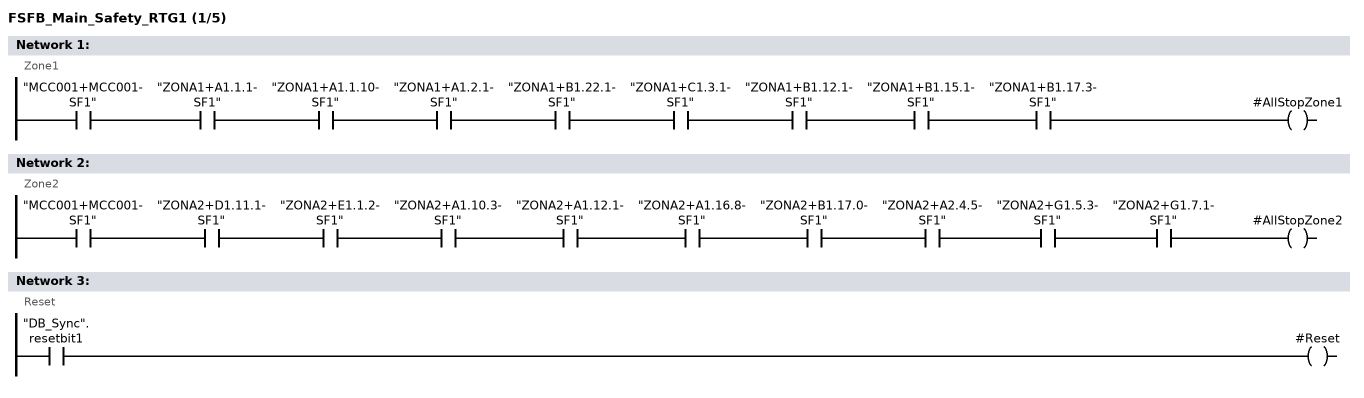
   RUNG wire#powerrail
      Contact( "MCC001+MCC001-SF1" )
      Contact( "ZONA1+A1.1.1-SF1" )
      Contact( "ZONA1+A1.1.10-SF1" )
      Contact( "ZONA1+A1.2.1-SF1" )
      Contact( "ZONA1+B1.22.1-SF1" )
      Contact( "ZONA1+C1.3.1-SF1" )
      Contact( "ZONA1+B1.12.1-SF1" )
      Contact( "ZONA1+B1.15.1-SF1" )
      Contact( "ZONA1+B1.17.3-SF1" )
      Coil( #AllStopZone1 )
   END_RUNG
   // the same network as SCL:
   #AllStopZone1 := "MCC001+MCC001-SF1" AND "ZONA1+A1.1.1-SF1" AND "ZONA1+A1.1.10-SF1" AND "ZONA1+A1.2.1-SF1" AND "ZONA1+B1.22.1-SF1" AND "ZONA1+C1.3.1-SF1" AND "ZONA1+B1.12.1-SF1" AND "ZONA1+B1.15.1-SF1" AND "ZONA1+B1.17.3-SF1";
END_REGION

REGION Network 2
   // Zone2
   RUNG wire#powerrail
      Contact( "MCC001+MCC001-SF1" )
      Contact( "ZONA2+D1.11.1-SF1" )
      Contact( "ZONA2+E1.1.2-SF1" )
      Contact( "ZONA2+A1.10.3-SF1" )
      Contact( "ZONA2+A1.12.1-SF1" )
      Contact( "ZONA2+A1.16.8-SF1" )
      Contact( "ZONA2+B1.17.0-SF1" )
      Contact( "ZONA2+A2.4.5-SF1" )
      Contact( "ZONA2+G1.5.3-SF1" )
      Contact( "ZONA2+G1.7.1-SF1" )
      Coil( #AllStopZone2 )
   END_RUNG
   // the same network as SCL:
   #AllStopZone2 := "MCC001+MCC001-SF1" AND "ZONA2+D1.11.1-SF1" AND "ZONA2+E1.1.2-SF1" AND "ZONA2+A1.10.3-SF1" AND "ZONA2+A1.12.1-SF1" AND "ZONA2+A1.16.8-SF1" AND "ZONA2+B1.17.0-SF1" AND "ZONA2+A2.4.5-SF1" AND "ZONA2+G1.5.3-SF1" AND "ZONA2+G1.7.1-SF1";
END_REGION

REGION Network 3
   // Reset
   RUNG wire#powerrail
      Contact( "DB_Sync".resetbit1 )
      Coil( #Reset )
   END_RUNG
   // the same network as SCL:
   #Reset := "DB_Sync".resetbit1;
END_REGION

REGION Network 4
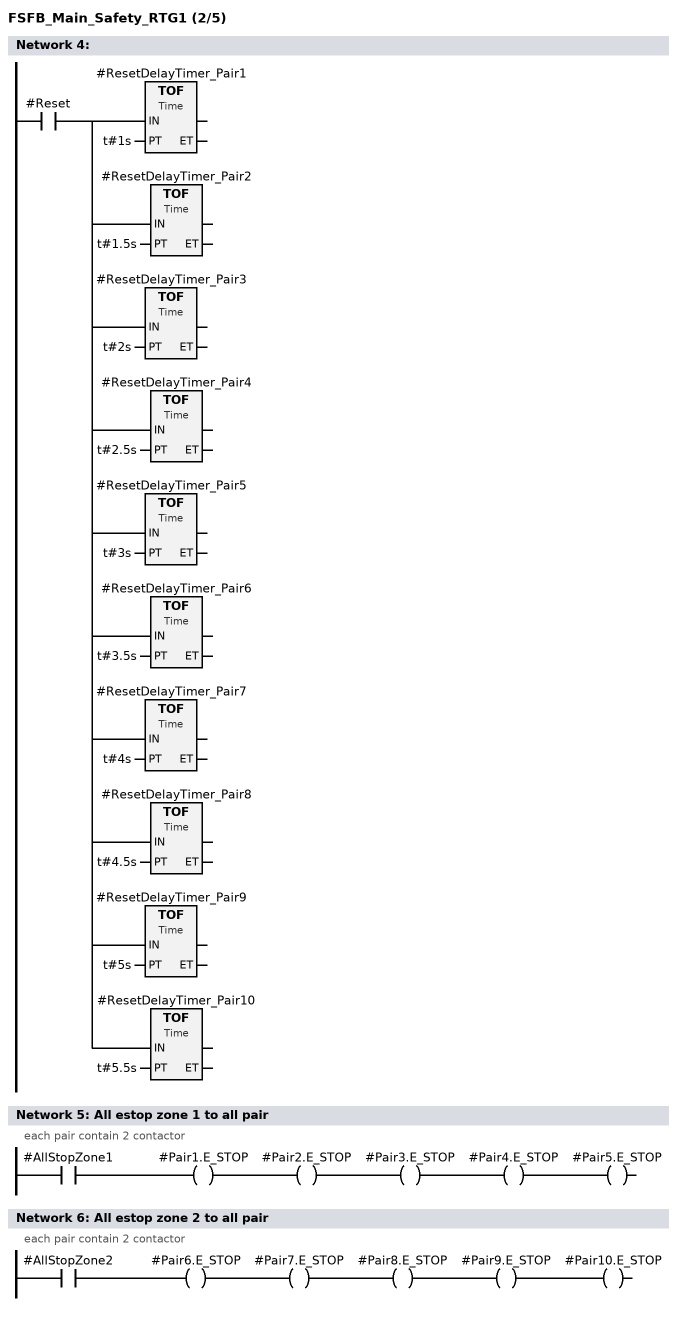
   RUNG wire#powerrail
      Contact( #Reset )
      wire#w1
      { S7_Templates := "[time_type := Time, codedbool_type := DInt]" } #ResetDelayTimer_Pair1.TOF(pt := t#1s, et =>)
   END_RUNG
   RUNG wire#w1
      { S7_Templates := "[time_type := Time, codedbool_type := DInt]" } #ResetDelayTimer_Pair2.TOF(pt := t#1.5s, et =>)
   END_RUNG
   RUNG wire#w1
      { S7_Templates := "[time_type := Time, codedbool_type := DInt]" } #ResetDelayTimer_Pair3.TOF(pt := t#2s, et =>)
   END_RUNG
   RUNG wire#w1
      { S7_Templates := "[time_type := Time, codedbool_type := DInt]" } #ResetDelayTimer_Pair4.TOF(pt := t#2.5s, et =>)
   END_RUNG
   RUNG wire#w1
      { S7_Templates := "[time_type := Time, codedbool_type := DInt]" } #ResetDelayTimer_Pair5.TOF(pt := t#3s, et =>)
   END_RUNG
   RUNG wire#w1
      { S7_Templates := "[time_type := Time, codedbool_type := DInt]" } #ResetDelayTimer_Pair6.TOF(pt := t#3.5s, et =>)
   END_RUNG
   RUNG wire#w1
      { S7_Templates := "[time_type := Time, codedbool_type := DInt]" } #ResetDelayTimer_Pair7.TOF(pt := t#4s, et =>)
   END_RUNG
   RUNG wire#w1
      { S7_Templates := "[time_type := Time, codedbool_type := DInt]" } #ResetDelayTimer_Pair8.TOF(pt := t#4.5s, et =>)
   END_RUNG
   RUNG wire#w1
      { S7_Templates := "[time_type := Time, codedbool_type := DInt]" } #ResetDelayTimer_Pair9.TOF(pt := t#5s, et =>)
   END_RUNG
   RUNG wire#w1
      { S7_Templates := "[time_type := Time, codedbool_type := DInt]" } #ResetDelayTimer_Pair10.TOF(pt := t#5.5s, et =>)
   END_RUNG
   // the same network as SCL:
   #ResetDelayTimer_Pair1.TOF(IN := #Reset, PT := t#1s);
   #ResetDelayTimer_Pair2.TOF(IN := #Reset, PT := t#1.5s);
   #ResetDelayTimer_Pair3.TOF(IN := #Reset, PT := t#2s);
   #ResetDelayTimer_Pair4.TOF(IN := #Reset, PT := t#2.5s);
   #ResetDelayTimer_Pair5.TOF(IN := #Reset, PT := t#3s);
   #ResetDelayTimer_Pair6.TOF(IN := #Reset, PT := t#3.5s);
   #ResetDelayTimer_Pair7.TOF(IN := #Reset, PT := t#4s);
   #ResetDelayTimer_Pair8.TOF(IN := #Reset, PT := t#4.5s);
   #ResetDelayTimer_Pair9.TOF(IN := #Reset, PT := t#5s);
   #ResetDelayTimer_Pair10.TOF(IN := #Reset, PT := t#5.5s);
END_REGION

REGION Network 5: All estop zone 1 to all pair
   // each pair contain 2 contactor
   RUNG wire#powerrail
      Contact( #AllStopZone1 )
      Coil( #Pair1.E_STOP )
      Coil( #Pair2.E_STOP )
      Coil( #Pair3.E_STOP )
      Coil( #Pair4.E_STOP )
      Coil( #Pair5.E_STOP )
   END_RUNG
   // the same network as SCL:
   #Pair1.E_STOP := #AllStopZone1;
   #Pair2.E_STOP := #AllStopZone1;
   #Pair3.E_STOP := #AllStopZone1;
   #Pair4.E_STOP := #AllStopZone1;
   #Pair5.E_STOP := #AllStopZone1;
END_REGION

REGION Network 6: All estop zone 2 to all pair
   // each pair contain 2 contactor
   RUNG wire#powerrail
      Contact( #AllStopZone2 )
      Coil( #Pair6.E_STOP )
      Coil( #Pair7.E_STOP )
      Coil( #Pair8.E_STOP )
      Coil( #Pair9.E_STOP )
      Coil( #Pair10.E_STOP )
   END_RUNG
   // the same network as SCL:
   #Pair6.E_STOP := #AllStopZone2;
   #Pair7.E_STOP := #AllStopZone2;
   #Pair8.E_STOP := #AllStopZone2;
   #Pair9.E_STOP := #AllStopZone2;
   #Pair10.E_STOP := #AllStopZone2;
END_REGION

REGION Network 7: Pair 1
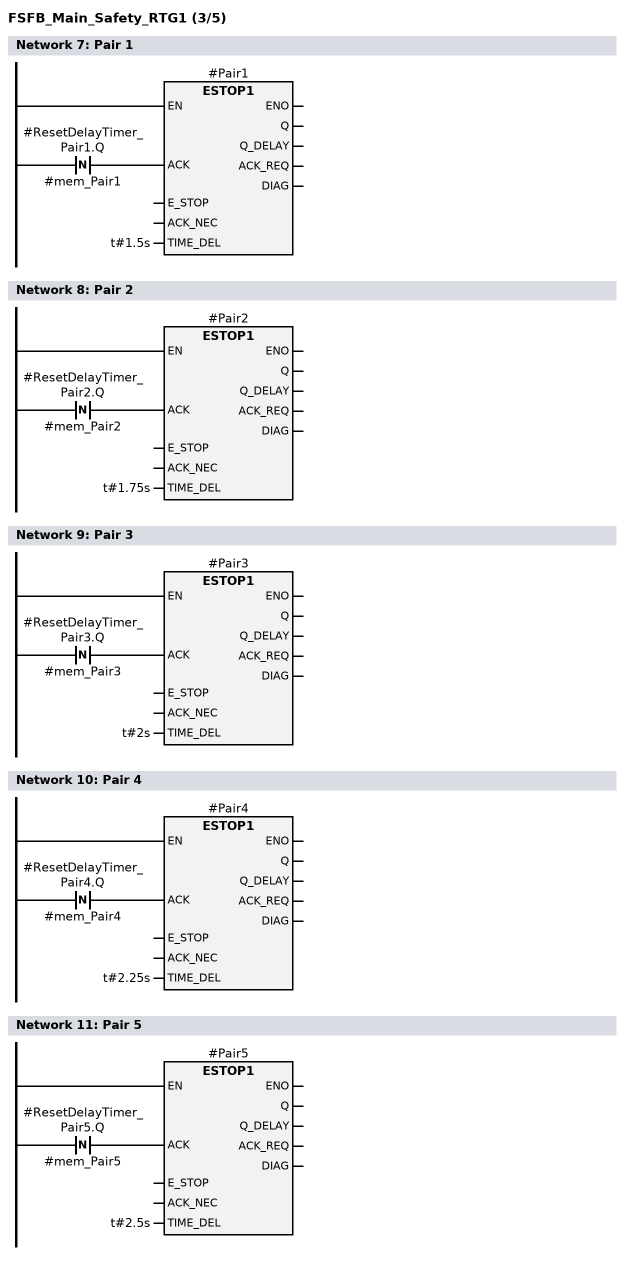
   RUNG wire#powerrail
      #Pair1.ESTOP1(ACK := wire#w1, E_STOP :=, ACK_NEC :=, TIME_DEL := t#1.5s, Q =>, Q_DELAY =>, ACK_REQ =>, DIAG =>)
   END_RUNG
   RUNG wire#powerrail
      N_Contact(operand := #ResetDelayTimer_Pair1.Q, bit := #mem_Pair1)
   END_RUNG wire#w1
   // the same network as SCL:
   #_w1 := NOT #ResetDelayTimer_Pair1.Q AND #mem_Pair1;   // falling edge of #ResetDelayTimer_Pair1.Q
   #mem_Pair1 := #ResetDelayTimer_Pair1.Q;
   #Pair1(ACK := #_w1, TIME_DEL := t#1.5s);   // ESTOP1
END_REGION

REGION Network 8: Pair 2
   RUNG wire#powerrail
      #Pair2.ESTOP1(ACK := wire#w1, E_STOP :=, ACK_NEC :=, TIME_DEL := t#1.75s, Q =>, Q_DELAY =>, ACK_REQ =>, DIAG =>)
   END_RUNG
   RUNG wire#powerrail
      N_Contact(operand := #ResetDelayTimer_Pair2.Q, bit := #mem_Pair2)
   END_RUNG wire#w1
   // the same network as SCL:
   #_w1 := NOT #ResetDelayTimer_Pair2.Q AND #mem_Pair2;   // falling edge of #ResetDelayTimer_Pair2.Q
   #mem_Pair2 := #ResetDelayTimer_Pair2.Q;
   #Pair2(ACK := #_w1, TIME_DEL := t#1.75s);   // ESTOP1
END_REGION

REGION Network 9: Pair 3
   RUNG wire#powerrail
      #Pair3.ESTOP1(ACK := wire#w1, E_STOP :=, ACK_NEC :=, TIME_DEL := t#2s, Q =>, Q_DELAY =>, ACK_REQ =>, DIAG =>)
   END_RUNG
   RUNG wire#powerrail
      N_Contact(operand := #ResetDelayTimer_Pair3.Q, bit := #mem_Pair3)
   END_RUNG wire#w1
   // the same network as SCL:
   #_w1 := NOT #ResetDelayTimer_Pair3.Q AND #mem_Pair3;   // falling edge of #ResetDelayTimer_Pair3.Q
   #mem_Pair3 := #ResetDelayTimer_Pair3.Q;
   #Pair3(ACK := #_w1, TIME_DEL := t#2s);   // ESTOP1
END_REGION

REGION Network 10: Pair 4
   RUNG wire#powerrail
      #Pair4.ESTOP1(ACK := wire#w1, E_STOP :=, ACK_NEC :=, TIME_DEL := t#2.25s, Q =>, Q_DELAY =>, ACK_REQ =>, DIAG =>)
   END_RUNG
   RUNG wire#powerrail
      N_Contact(operand := #ResetDelayTimer_Pair4.Q, bit := #mem_Pair4)
   END_RUNG wire#w1
   // the same network as SCL:
   #_w1 := NOT #ResetDelayTimer_Pair4.Q AND #mem_Pair4;   // falling edge of #ResetDelayTimer_Pair4.Q
   #mem_Pair4 := #ResetDelayTimer_Pair4.Q;
   #Pair4(ACK := #_w1, TIME_DEL := t#2.25s);   // ESTOP1
END_REGION

REGION Network 11: Pair 5
   RUNG wire#powerrail
      #Pair5.ESTOP1(ACK := wire#w1, E_STOP :=, ACK_NEC :=, TIME_DEL := t#2.5s, Q =>, Q_DELAY =>, ACK_REQ =>, DIAG =>)
   END_RUNG
   RUNG wire#powerrail
      N_Contact(operand := #ResetDelayTimer_Pair5.Q, bit := #mem_Pair5)
   END_RUNG wire#w1
   // the same network as SCL:
   #_w1 := NOT #ResetDelayTimer_Pair5.Q AND #mem_Pair5;   // falling edge of #ResetDelayTimer_Pair5.Q
   #mem_Pair5 := #ResetDelayTimer_Pair5.Q;
   #Pair5(ACK := #_w1, TIME_DEL := t#2.5s);   // ESTOP1
END_REGION

REGION Network 12: Pair 6
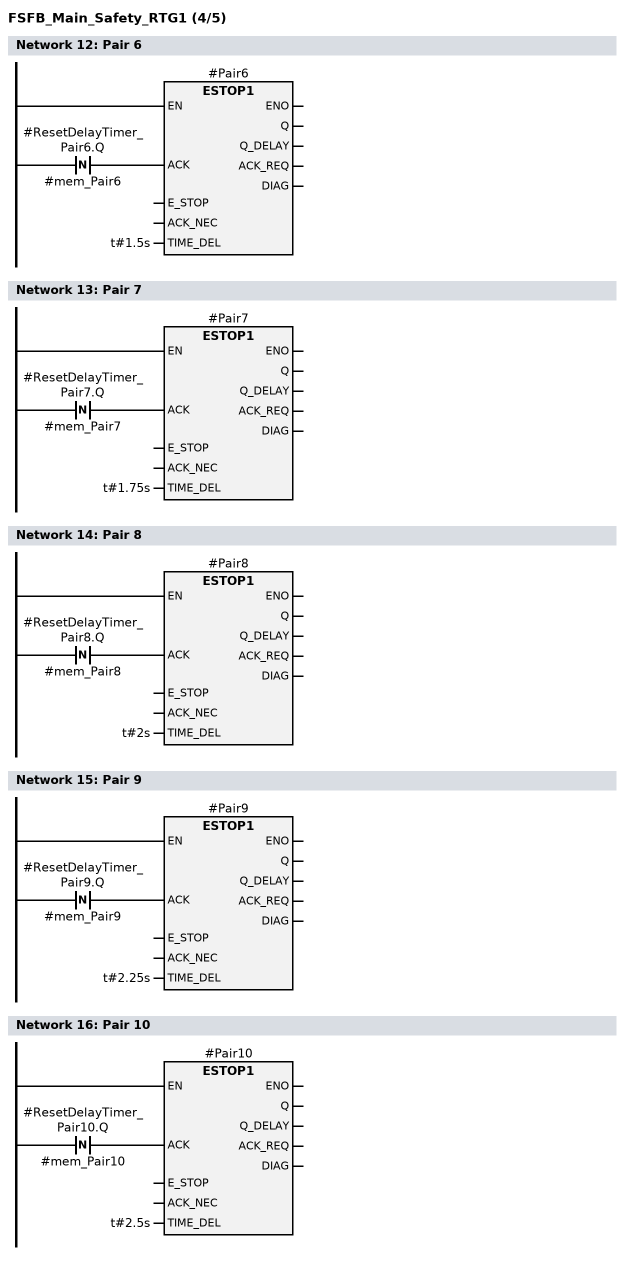
   RUNG wire#powerrail
      #Pair6.ESTOP1(ACK := wire#w1, E_STOP :=, ACK_NEC :=, TIME_DEL := t#1.5s, Q =>, Q_DELAY =>, ACK_REQ =>, DIAG =>)
   END_RUNG
   RUNG wire#powerrail
      N_Contact(operand := #ResetDelayTimer_Pair6.Q, bit := #mem_Pair6)
   END_RUNG wire#w1
   // the same network as SCL:
   #_w1 := NOT #ResetDelayTimer_Pair6.Q AND #mem_Pair6;   // falling edge of #ResetDelayTimer_Pair6.Q
   #mem_Pair6 := #ResetDelayTimer_Pair6.Q;
   #Pair6(ACK := #_w1, TIME_DEL := t#1.5s);   // ESTOP1
END_REGION

REGION Network 13: Pair 7
   RUNG wire#powerrail
      #Pair7.ESTOP1(ACK := wire#w1, E_STOP :=, ACK_NEC :=, TIME_DEL := t#1.75s, Q =>, Q_DELAY =>, ACK_REQ =>, DIAG =>)
   END_RUNG
   RUNG wire#powerrail
      N_Contact(operand := #ResetDelayTimer_Pair7.Q, bit := #mem_Pair7)
   END_RUNG wire#w1
   // the same network as SCL:
   #_w1 := NOT #ResetDelayTimer_Pair7.Q AND #mem_Pair7;   // falling edge of #ResetDelayTimer_Pair7.Q
   #mem_Pair7 := #ResetDelayTimer_Pair7.Q;
   #Pair7(ACK := #_w1, TIME_DEL := t#1.75s);   // ESTOP1
END_REGION

REGION Network 14: Pair 8
   RUNG wire#powerrail
      #Pair8.ESTOP1(ACK := wire#w1, E_STOP :=, ACK_NEC :=, TIME_DEL := t#2s, Q =>, Q_DELAY =>, ACK_REQ =>, DIAG =>)
   END_RUNG
   RUNG wire#powerrail
      N_Contact(operand := #ResetDelayTimer_Pair8.Q, bit := #mem_Pair8)
   END_RUNG wire#w1
   // the same network as SCL:
   #_w1 := NOT #ResetDelayTimer_Pair8.Q AND #mem_Pair8;   // falling edge of #ResetDelayTimer_Pair8.Q
   #mem_Pair8 := #ResetDelayTimer_Pair8.Q;
   #Pair8(ACK := #_w1, TIME_DEL := t#2s);   // ESTOP1
END_REGION

REGION Network 15: Pair 9
   RUNG wire#powerrail
      #Pair9.ESTOP1(ACK := wire#w1, E_STOP :=, ACK_NEC :=, TIME_DEL := t#2.25s, Q =>, Q_DELAY =>, ACK_REQ =>, DIAG =>)
   END_RUNG
   RUNG wire#powerrail
      N_Contact(operand := #ResetDelayTimer_Pair9.Q, bit := #mem_Pair9)
   END_RUNG wire#w1
   // the same network as SCL:
   #_w1 := NOT #ResetDelayTimer_Pair9.Q AND #mem_Pair9;   // falling edge of #ResetDelayTimer_Pair9.Q
   #mem_Pair9 := #ResetDelayTimer_Pair9.Q;
   #Pair9(ACK := #_w1, TIME_DEL := t#2.25s);   // ESTOP1
END_REGION

REGION Network 16: Pair 10
   RUNG wire#powerrail
      #Pair10.ESTOP1(ACK := wire#w1, E_STOP :=, ACK_NEC :=, TIME_DEL := t#2.5s, Q =>, Q_DELAY =>, ACK_REQ =>, DIAG =>)
   END_RUNG
   RUNG wire#powerrail
      N_Contact(operand := #ResetDelayTimer_Pair10.Q, bit := #mem_Pair10)
   END_RUNG wire#w1
   // the same network as SCL:
   #_w1 := NOT #ResetDelayTimer_Pair10.Q AND #mem_Pair10;   // falling edge of #ResetDelayTimer_Pair10.Q
   #mem_Pair10 := #ResetDelayTimer_Pair10.Q;
   #Pair10(ACK := #_w1, TIME_DEL := t#2.5s);   // ESTOP1
END_REGION

REGION Network 17: Output contactors
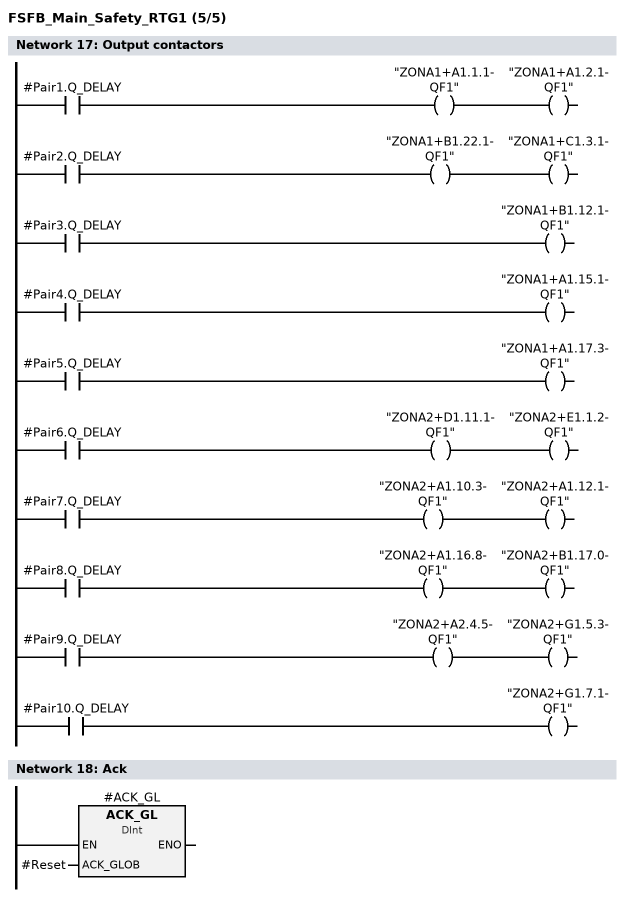
   RUNG wire#powerrail
      Contact( #Pair1.Q_DELAY )
      Coil( "ZONA1+A1.1.1-QF1" )
      Coil( "ZONA1+A1.2.1-QF1" )
   END_RUNG
   RUNG wire#powerrail
      Contact( #Pair2.Q_DELAY )
      Coil( "ZONA1+B1.22.1-QF1" )
      Coil( "ZONA1+C1.3.1-QF1" )
   END_RUNG
   RUNG wire#powerrail
      Contact( #Pair3.Q_DELAY )
      Coil( "ZONA1+B1.12.1-QF1" )
   END_RUNG
   RUNG wire#powerrail
      Contact( #Pair4.Q_DELAY )
      Coil( "ZONA1+A1.15.1-QF1" )
   END_RUNG
   RUNG wire#powerrail
      Contact( #Pair5.Q_DELAY )
      Coil( "ZONA1+A1.17.3-QF1" )
   END_RUNG
   RUNG wire#powerrail
      Contact( #Pair6.Q_DELAY )
      Coil( "ZONA2+D1.11.1-QF1" )
      Coil( "ZONA2+E1.1.2-QF1" )
   END_RUNG
   RUNG wire#powerrail
      Contact( #Pair7.Q_DELAY )
      Coil( "ZONA2+A1.10.3-QF1" )
      Coil( "ZONA2+A1.12.1-QF1" )
   END_RUNG
   RUNG wire#powerrail
      Contact( #Pair8.Q_DELAY )
      Coil( "ZONA2+A1.16.8-QF1" )
      Coil( "ZONA2+B1.17.0-QF1" )
   END_RUNG
   RUNG wire#powerrail
      Contact( #Pair9.Q_DELAY )
      Coil( "ZONA2+A2.4.5-QF1" )
      Coil( "ZONA2+G1.5.3-QF1" )
   END_RUNG
   RUNG wire#powerrail
      Contact( #Pair10.Q_DELAY )
      Coil( "ZONA2+G1.7.1-QF1" )
   END_RUNG
   // the same network as SCL:
   "ZONA1+A1.1.1-QF1" := #Pair1.Q_DELAY;
   "ZONA1+A1.2.1-QF1" := #Pair1.Q_DELAY;
   "ZONA1+B1.22.1-QF1" := #Pair2.Q_DELAY;
   "ZONA1+C1.3.1-QF1" := #Pair2.Q_DELAY;
   "ZONA1+B1.12.1-QF1" := #Pair3.Q_DELAY;
   "ZONA1+A1.15.1-QF1" := #Pair4.Q_DELAY;
   "ZONA1+A1.17.3-QF1" := #Pair5.Q_DELAY;
   "ZONA2+D1.11.1-QF1" := #Pair6.Q_DELAY;
   "ZONA2+E1.1.2-QF1" := #Pair6.Q_DELAY;
   "ZONA2+A1.10.3-QF1" := #Pair7.Q_DELAY;
   "ZONA2+A1.12.1-QF1" := #Pair7.Q_DELAY;
   "ZONA2+A1.16.8-QF1" := #Pair8.Q_DELAY;
   "ZONA2+B1.17.0-QF1" := #Pair8.Q_DELAY;
   "ZONA2+A2.4.5-QF1" := #Pair9.Q_DELAY;
   "ZONA2+G1.5.3-QF1" := #Pair9.Q_DELAY;
   "ZONA2+G1.7.1-QF1" := #Pair10.Q_DELAY;
END_REGION

REGION Network 18: Ack
   RUNG wire#powerrail
      { S7_Templates := "codedbool_type := DInt" } #ACK_GL.ACK_GL(ACK_GLOB := #Reset)
   END_RUNG
   // the same network as SCL:
   #ACK_GL(ACK_GLOB := #Reset);   // ACK_GL
END_REGION
END_FUNCTION_BLOCK

FUNCTION_BLOCK "FB_AutoReset"   // FB21, LAD
// stored: Access Published, MemoryReserve 100, Namespace Global, SetENOAutomatically false
   VAR_INPUT
      AckIN : Bool;
   END_VAR
   VAR_OUTPUT
      Ack : Bool;
   END_VAR
   VAR
      MemoryBit : Array[1..2] of Bool;
      "Timer" { S7_SetPoint := 'True'} : TOF_TIME;
   END_VAR
   VAR_TEMP   // added for the SCL form of the ladder/FBD networks
      _w1 : Bool;
      _w2 : Bool;
   END_VAR
BEGIN

REGION Network 1
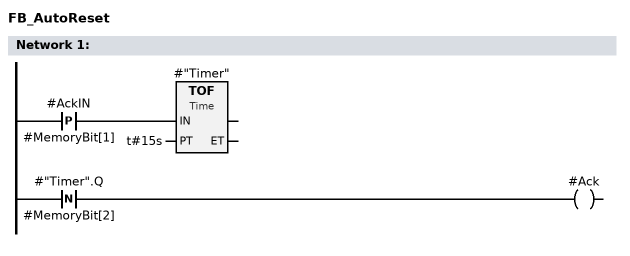
   RUNG wire#powerrail
      P_Contact(operand := #AckIN, bit := #MemoryBit[1])
      { S7_Templates := "time_type := Time" } #"Timer".TOF(pt := t#15s, et =>)
   END_RUNG
   RUNG wire#powerrail
      N_Contact(operand := #"Timer".Q, bit := #MemoryBit[2])
      Coil( #Ack )
   END_RUNG
   // the same network as SCL:
   #_w1 := #AckIN AND NOT #MemoryBit[1];   // rising edge of #AckIN
   #MemoryBit[1] := #AckIN;
   #"Timer"(IN := #_w1, PT := t#15s);   // TOF
   #_w2 := NOT #"Timer".Q AND #MemoryBit[2];   // falling edge of #"Timer".Q
   #MemoryBit[2] := #"Timer".Q;
   #Ack := #_w2;
END_REGION
END_FUNCTION_BLOCK

FUNCTION_BLOCK "FB_ManualControl"   // FB37, LAD
// stored: Access Published, MemoryReserve 100, Namespace Global, SetENOAutomatically false
   VAR RETAIN
      "Counter" { S7_SetPoint := 'True'} : CTU_INT;
   END_VAR
BEGIN

REGION Network 1
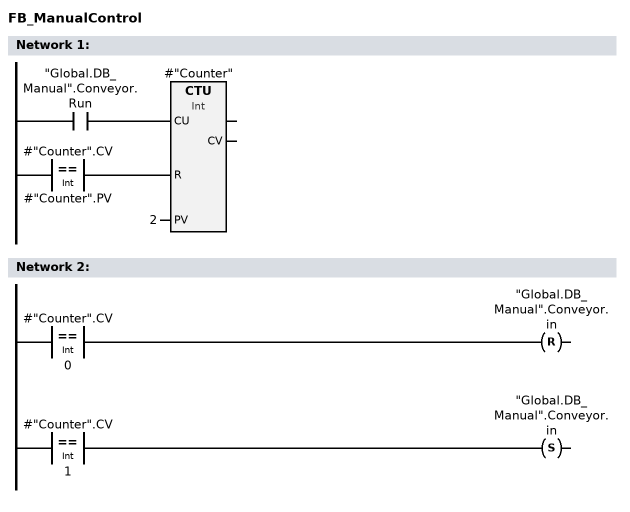
   RUNG wire#powerrail
      Contact( "Global.DB_Manual".Conveyor.Run )
      { S7_Templates := "value_type := Int" } #"Counter".CTU(r := wire#w1, pv := 2, cv =>)
   END_RUNG
   RUNG wire#powerrail
      { S7_Templates := "SrcType := Int" } EQ_Contact(in1 := #"Counter".CV, in2 := #"Counter".PV)
   END_RUNG wire#w1
   // the same network as SCL:
   #"Counter"(CU := "Global.DB_Manual".Conveyor.Run, R := #"Counter".CV = #"Counter".PV, PV := 2);   // CTU
END_REGION

REGION Network 2
   RUNG wire#powerrail
      { S7_Templates := "SrcType := Int" } EQ_Contact(in1 := #"Counter".CV, in2 := 0)
      R_Coil( "Global.DB_Manual".Conveyor.in )
   END_RUNG
   RUNG wire#powerrail
      { S7_Templates := "SrcType := Int" } EQ_Contact(in1 := #"Counter".CV, in2 := 1)
      S_Coil( "Global.DB_Manual".Conveyor.in )
   END_RUNG
   // the same network as SCL:
   IF #"Counter".CV = 0 THEN "Global.DB_Manual".Conveyor.in := FALSE; END_IF;
   IF #"Counter".CV = 1 THEN "Global.DB_Manual".Conveyor.in := TRUE; END_IF;
END_REGION
END_FUNCTION_BLOCK

FUNCTION "FC_ManualSorter" : Void   // FC18, LAD
// stored: Access Published, Namespace Global, SetENOAutomatically false
   VAR_INPUT
      RunWheels : Bool;
      "GoRight/left" : Bool;
      GoStraight : Bool;
      "positionRight/Left" : Bool;
      positionStraight : Bool;
   END_VAR
   VAR_OUTPUT
      CmdRunWheels : Bool;
      "CmdRight/Left" : Bool;
      CmdStraight : Bool;
   END_VAR
BEGIN

REGION Network 1: status manual
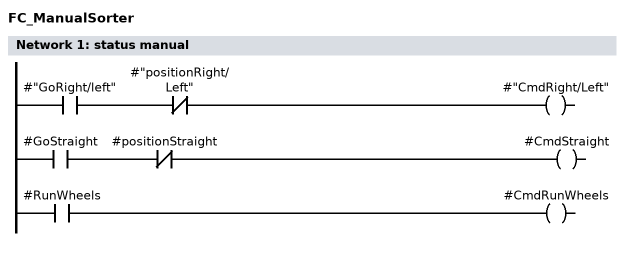
   RUNG wire#powerrail
      Contact( #"GoRight/left" )
      I_Contact( #"positionRight/Left" )
      Coil( #"CmdRight/Left" )
   END_RUNG
   RUNG wire#powerrail
      Contact( #GoStraight )
      I_Contact( #positionStraight )
      Coil( #CmdStraight )
   END_RUNG
   RUNG wire#powerrail
      Contact( #RunWheels )
      Coil( #CmdRunWheels )
   END_RUNG
   // the same network as SCL:
   #"CmdRight/Left" := #"GoRight/left" AND NOT #"positionRight/Left";
   #CmdStraight := #GoStraight AND NOT #positionStraight;
   #CmdRunWheels := #RunWheels;
END_REGION
END_FUNCTION

FUNCTION "FC_ManualStopper" : Void   // FC13, LAD
// stored: Access Published, Namespace Global, SetENOAutomatically false
   VAR_INPUT
      GoUp : Bool;
      GoDown : Bool;
      positionUp : Bool;
      positionDown : Bool;
   END_VAR
   VAR_OUTPUT
      CmdUP : Bool;
      cmdDOWN : Bool;
   END_VAR
BEGIN

REGION Network 1: status manual
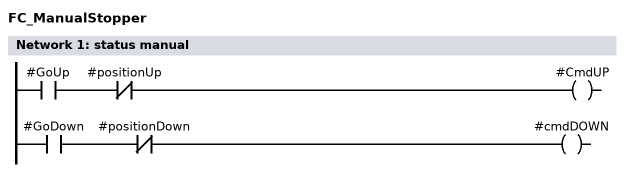
   RUNG wire#powerrail
      Contact( #GoUp )
      I_Contact( #positionUp )
      Coil( #CmdUP )
   END_RUNG
   RUNG wire#powerrail
      Contact( #GoDown )
      I_Contact( #positionDown )
      Coil( #cmdDOWN )
   END_RUNG
   // the same network as SCL:
   #CmdUP := #GoUp AND NOT #positionUp;
   #cmdDOWN := #GoDown AND NOT #positionDown;
END_REGION
END_FUNCTION

FUNCTION_BLOCK "FB_MABS_PNIO"   // FB6, LAD
// stored: Access Published, MemoryReserve 100, Namespace Global, SetENOAutomatically false
   VAR_IN_OUT
      IBP_in : "Global.IB_P01_02_03_in_64bytes_struct";
      IBP_out : "Global.IB_P01_02_03_out_64bytes_struct";
      MABS : "Global.MABS";
   END_VAR
   VAR
      Initializing : Bool;
      Waiting_sw_req : Bool;
      Switching_left : Bool;
      "Switching_left to straight" : Bool;
      "Switching_right to straight" : Bool;
      Switching_right : Bool;
      Switching_done : Bool;
      Tof_life_bit { S7_SetPoint := 'True'} : TON_TIME;
      MABS_sw_timout { S7_SetPoint := 'True'} : TON_TIME;
      "position status_right" : Bool;
      "position status_left" : Bool;
      "position status_straight" : Bool;
      Edge0 : Bool;
      Edge1 : Bool;
      Edge2 : Bool;
      Edge3 : Bool;
      Edge4 : Bool;
      Edge5 : Bool;
      Edge6 : Bool;
      Ton_err_motor_A { S7_SetPoint := 'True'} : TON_TIME;
      Ton_err_motor_B { S7_SetPoint := 'True'} : TON_TIME;
      Ton_err_motor_Com { S7_SetPoint := 'True'} : TON_TIME;
   END_VAR
   VAR_TEMP
      Temp_err_com : Bool;
   END_VAR
   VAR_TEMP   // added for the SCL form of the ladder/FBD networks
      _w1 : Bool;
      _w2 : Bool;
   END_VAR
BEGIN

REGION Network 1: Error motor A & B
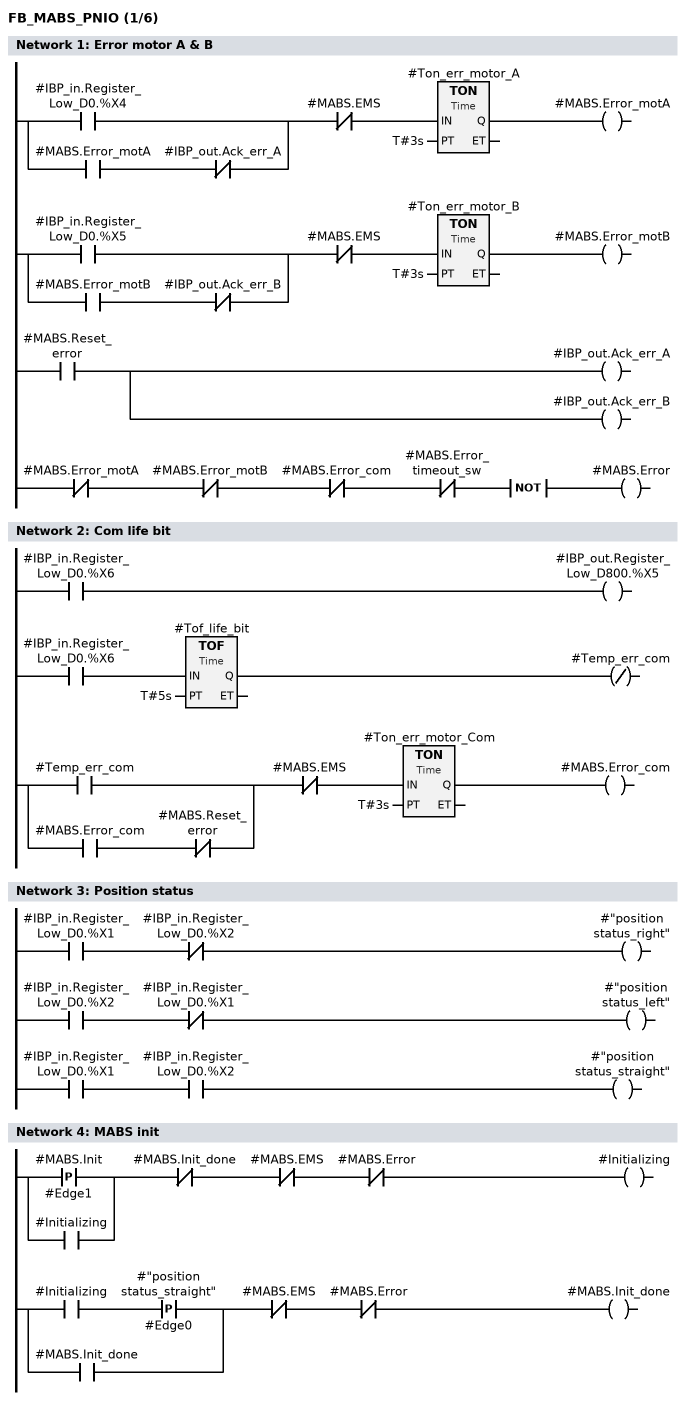
   RUNG wire#powerrail
      Contact( #IBP_in.Register_Low_D0.%X4 )
      wire#w1
      I_Contact( #MABS.EMS )
      { S7_Templates := "time_type := Time" } #Ton_err_motor_A.TON(pt := T#3s, et =>)
      Coil( #MABS.Error_motA )
   END_RUNG
   RUNG wire#powerrail
      Contact( #MABS.Error_motA )
      I_Contact( #IBP_out.Ack_err_A )
   END_RUNG wire#w1
   RUNG wire#powerrail
      Contact( #IBP_in.Register_Low_D0.%X5 )
      wire#w2
      I_Contact( #MABS.EMS )
      { S7_Templates := "time_type := Time" } #Ton_err_motor_B.TON(pt := T#3s, et =>)
      Coil( #MABS.Error_motB )
   END_RUNG
   RUNG wire#powerrail
      Contact( #MABS.Error_motB )
      I_Contact( #IBP_out.Ack_err_B )
   END_RUNG wire#w2
   RUNG wire#powerrail
      Contact( #MABS.Reset_error )
      wire#w3
      Coil( #IBP_out.Ack_err_A )
   END_RUNG
   RUNG wire#w3
      Coil( #IBP_out.Ack_err_B )
   END_RUNG
   RUNG wire#powerrail
      I_Contact( #MABS.Error_motA )
      I_Contact( #MABS.Error_motB )
      I_Contact( #MABS.Error_com )
      I_Contact( #MABS.Error_timeout_sw )
      Not()
      Coil( #MABS.Error )
   END_RUNG
   // the same network as SCL:
   #Ton_err_motor_A(IN := (#IBP_in.Register_Low_D0.%X4 OR (#MABS.Error_motA AND NOT #IBP_out.Ack_err_A)) AND NOT #MABS.EMS,   // TON
                    PT := T#3s);
   #MABS.Error_motA := #Ton_err_motor_A.Q;
   #Ton_err_motor_B(IN := (#IBP_in.Register_Low_D0.%X5 OR (#MABS.Error_motB AND NOT #IBP_out.Ack_err_B)) AND NOT #MABS.EMS,   // TON
                    PT := T#3s);
   #MABS.Error_motB := #Ton_err_motor_B.Q;
   #IBP_out.Ack_err_A := #MABS.Reset_error;
   #IBP_out.Ack_err_B := #MABS.Reset_error;
   #MABS.Error := NOT (NOT #MABS.Error_motA AND NOT #MABS.Error_motB AND NOT #MABS.Error_com AND NOT #MABS.Error_timeout_sw);
END_REGION

REGION Network 2: Com life bit
   RUNG wire#powerrail
      Contact( #IBP_in.Register_Low_D0.%X6 )
      Coil( #IBP_out.Register_Low_D800.%X5 )
   END_RUNG
   RUNG wire#powerrail
      Contact( #IBP_in.Register_Low_D0.%X6 )
      { S7_Templates := "time_type := Time" } #Tof_life_bit.TOF(pt := T#5s, et =>)
      I_Coil( #Temp_err_com )
   END_RUNG
   RUNG wire#powerrail
      Contact( #Temp_err_com )
      wire#w1
      I_Contact( #MABS.EMS )
      { S7_Templates := "time_type := Time" } #Ton_err_motor_Com.TON(pt := T#3s, et =>)
      Coil( #MABS.Error_com )
   END_RUNG
   RUNG wire#powerrail
      Contact( #MABS.Error_com )
      I_Contact( #MABS.Reset_error )
   END_RUNG wire#w1
   // the same network as SCL:
   #IBP_out.Register_Low_D800.%X5 := #IBP_in.Register_Low_D0.%X6;
   #Tof_life_bit(IN := #IBP_in.Register_Low_D0.%X6, PT := T#5s);   // TOF
   #Temp_err_com := NOT #Tof_life_bit.Q;
   #Ton_err_motor_Com(IN := (#Temp_err_com OR (#MABS.Error_com AND NOT #MABS.Reset_error)) AND NOT #MABS.EMS,   // TON
                      PT := T#3s);
   #MABS.Error_com := #Ton_err_motor_Com.Q;
END_REGION

REGION Network 3: Position status
   RUNG wire#powerrail
      Contact( #IBP_in.Register_Low_D0.%X1 )
      I_Contact( #IBP_in.Register_Low_D0.%X2 )
      Coil( #"position status_right" )
   END_RUNG
   RUNG wire#powerrail
      Contact( #IBP_in.Register_Low_D0.%X2 )
      I_Contact( #IBP_in.Register_Low_D0.%X1 )
      Coil( #"position status_left" )
   END_RUNG
   RUNG wire#powerrail
      Contact( #IBP_in.Register_Low_D0.%X1 )
      Contact( #IBP_in.Register_Low_D0.%X2 )
      Coil( #"position status_straight" )
   END_RUNG
   // the same network as SCL:
   #"position status_right" := #IBP_in.Register_Low_D0.%X1 AND NOT #IBP_in.Register_Low_D0.%X2;
   #"position status_left" := #IBP_in.Register_Low_D0.%X2 AND NOT #IBP_in.Register_Low_D0.%X1;
   #"position status_straight" := #IBP_in.Register_Low_D0.%X1 AND #IBP_in.Register_Low_D0.%X2;
END_REGION

REGION Network 4: MABS init
   RUNG wire#powerrail
      P_Contact(operand := #MABS.Init, bit := #Edge1)
      wire#w1
      I_Contact( #MABS.Init_done )
      I_Contact( #MABS.EMS )
      I_Contact( #MABS.Error )
      Coil( #Initializing )
   END_RUNG
   RUNG wire#powerrail
      Contact( #Initializing )
   END_RUNG wire#w1
   RUNG wire#powerrail
      Contact( #Initializing )
      P_Contact(operand := #"position status_straight", bit := #Edge0)
      wire#w2
      I_Contact( #MABS.EMS )
      I_Contact( #MABS.Error )
      Coil( #MABS.Init_done )
   END_RUNG
   RUNG wire#powerrail
      Contact( #MABS.Init_done )
   END_RUNG wire#w2
   // the same network as SCL:
   #_w1 := #MABS.Init AND NOT #Edge1;   // rising edge of #MABS.Init
   #Edge1 := #MABS.Init;
   #Initializing := (#_w1 OR #Initializing) AND NOT #MABS.Init_done AND NOT #MABS.EMS AND NOT #MABS.Error;
   #_w2 := #Initializing AND #"position status_straight" AND NOT #Edge0;   // rising edge of #"position status_straight"
   #Edge0 := #"position status_straight";
   #MABS.Init_done := (#_w2 OR #MABS.Init_done) AND NOT #MABS.EMS AND NOT #MABS.Error;
END_REGION

REGION Network 5: MABS ready
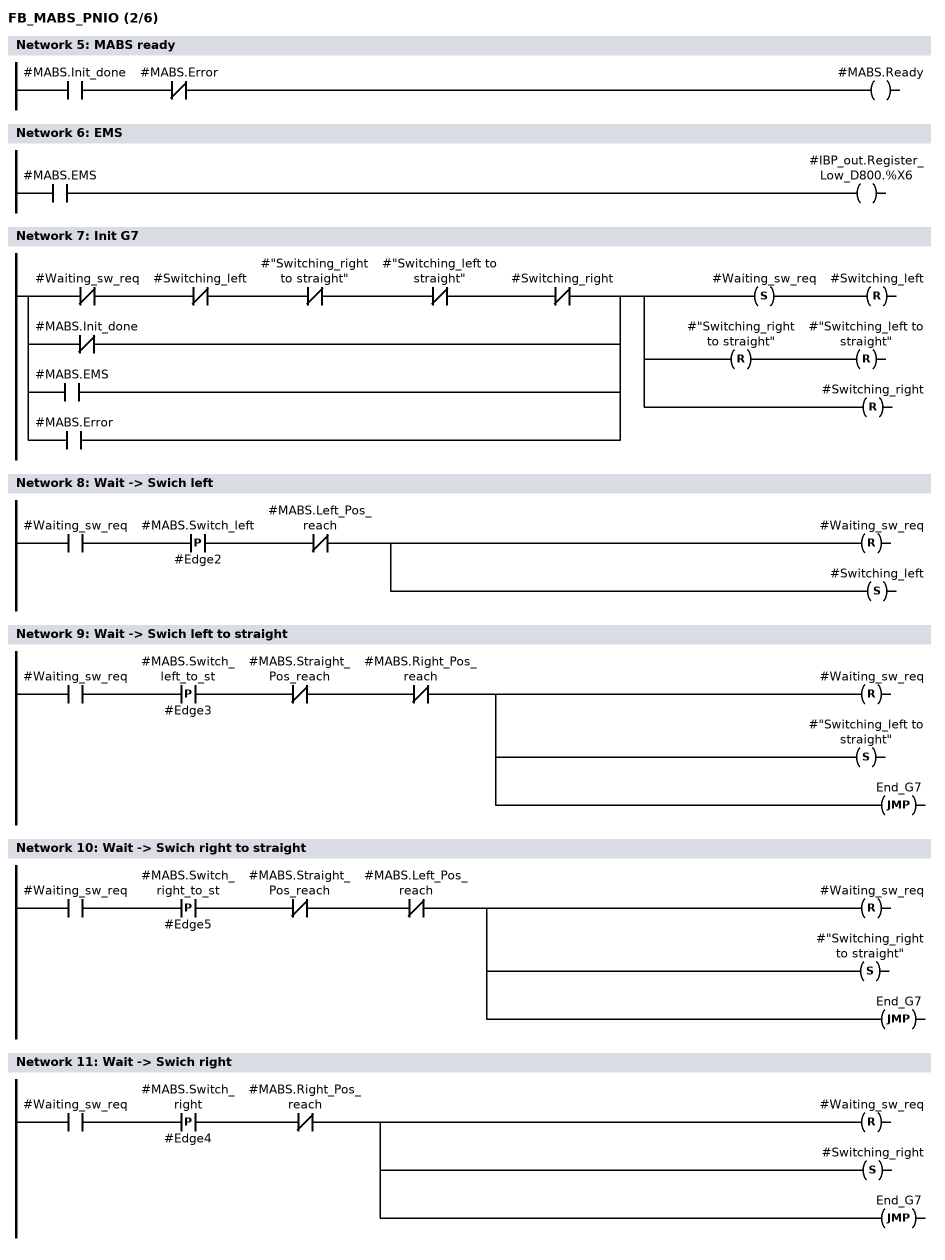
   RUNG wire#powerrail
      Contact( #MABS.Init_done )
      I_Contact( #MABS.Error )
      Coil( #MABS.Ready )
   END_RUNG
   // the same network as SCL:
   #MABS.Ready := #MABS.Init_done AND NOT #MABS.Error;
END_REGION

REGION Network 6: EMS
   RUNG wire#powerrail
      Contact( #MABS.EMS )
      Coil( #IBP_out.Register_Low_D800.%X6 )
   END_RUNG
   // the same network as SCL:
   #IBP_out.Register_Low_D800.%X6 := #MABS.EMS;
END_REGION

REGION Network 7: Init G7
   RUNG wire#powerrail
      I_Contact( #Waiting_sw_req )
      I_Contact( #Switching_left )
      I_Contact( #"Switching_right to straight" )
      I_Contact( #"Switching_left to straight" )
      I_Contact( #Switching_right )
      wire#w1
      S_Coil( #Waiting_sw_req )
      R_Coil( #Switching_left )
   END_RUNG
   RUNG wire#powerrail
      I_Contact( #MABS.Init_done )
   END_RUNG wire#w1
   RUNG wire#powerrail
      Contact( #MABS.EMS )
   END_RUNG wire#w1
   RUNG wire#powerrail
      Contact( #MABS.Error )
   END_RUNG wire#w1
   RUNG wire#w1
      R_Coil( #"Switching_right to straight" )
      R_Coil( #"Switching_left to straight" )
   END_RUNG
   RUNG wire#w1
      R_Coil( #Switching_right )
   END_RUNG
   // the same network as SCL:
   #_w1 := (NOT #Waiting_sw_req AND NOT #Switching_left AND NOT #"Switching_right to straight" AND NOT #"Switching_left to straight" AND NOT #Switching_right) OR NOT #MABS.Init_done OR #MABS.EMS OR #MABS.Error;
   IF #_w1 THEN
       #Waiting_sw_req := TRUE;
       #Switching_left := FALSE;
       #"Switching_right to straight" := FALSE;
       #"Switching_left to straight" := FALSE;
       #Switching_right := FALSE;
   END_IF;
END_REGION

REGION Network 8: Wait -> Swich left
   RUNG wire#powerrail
      Contact( #Waiting_sw_req )
      P_Contact(operand := #MABS.Switch_left, bit := #Edge2)
      I_Contact( #MABS.Left_Pos_reach )
      wire#w1
      R_Coil( #Waiting_sw_req )
   END_RUNG
   RUNG wire#w1
      S_Coil( #Switching_left )
   END_RUNG
   // the same network as SCL:
   #_w1 := #Waiting_sw_req AND #MABS.Switch_left AND NOT #Edge2;   // rising edge of #MABS.Switch_left
   #Edge2 := #MABS.Switch_left;
   IF #_w1 AND NOT #MABS.Left_Pos_reach THEN
       #Waiting_sw_req := FALSE;
       #Switching_left := TRUE;
   END_IF;
END_REGION

REGION Network 9: Wait -> Swich left to straight
   RUNG wire#powerrail
      Contact( #Waiting_sw_req )
      P_Contact(operand := #MABS.Switch_left_to_st, bit := #Edge3)
      I_Contact( #MABS.Straight_Pos_reach )
      I_Contact( #MABS.Right_Pos_reach )
      wire#w1
      R_Coil( #Waiting_sw_req )
   END_RUNG
   RUNG wire#w1
      S_Coil( #"Switching_left to straight" )
   END_RUNG
   RUNG wire#w1
      JumpCoil( End_G7 )
   END_RUNG
   // the same network as SCL:
   #_w1 := #Waiting_sw_req AND #MABS.Switch_left_to_st AND NOT #Edge3;   // rising edge of #MABS.Switch_left_to_st
   #Edge3 := #MABS.Switch_left_to_st;
   #_w2 := #_w1 AND NOT #MABS.Straight_Pos_reach AND NOT #MABS.Right_Pos_reach;
   IF #_w2 THEN
       #Waiting_sw_req := FALSE;
       #"Switching_left to straight" := TRUE;
       GOTO End_G7;
   END_IF;
END_REGION

REGION Network 10: Wait -> Swich right to straight
   RUNG wire#powerrail
      Contact( #Waiting_sw_req )
      P_Contact(operand := #MABS.Switch_right_to_st, bit := #Edge5)
      I_Contact( #MABS.Straight_Pos_reach )
      I_Contact( #MABS.Left_Pos_reach )
      wire#w1
      R_Coil( #Waiting_sw_req )
   END_RUNG
   RUNG wire#w1
      S_Coil( #"Switching_right to straight" )
   END_RUNG
   RUNG wire#w1
      JumpCoil( End_G7 )
   END_RUNG
   // the same network as SCL:
   #_w1 := #Waiting_sw_req AND #MABS.Switch_right_to_st AND NOT #Edge5;   // rising edge of #MABS.Switch_right_to_st
   #Edge5 := #MABS.Switch_right_to_st;
   #_w2 := #_w1 AND NOT #MABS.Straight_Pos_reach AND NOT #MABS.Left_Pos_reach;
   IF #_w2 THEN
       #Waiting_sw_req := FALSE;
       #"Switching_right to straight" := TRUE;
       GOTO End_G7;
   END_IF;
END_REGION

REGION Network 11: Wait -> Swich right
   RUNG wire#powerrail
      Contact( #Waiting_sw_req )
      P_Contact(operand := #MABS.Switch_right, bit := #Edge4)
      I_Contact( #MABS.Right_Pos_reach )
      wire#w1
      R_Coil( #Waiting_sw_req )
   END_RUNG
   RUNG wire#w1
      S_Coil( #Switching_right )
   END_RUNG
   RUNG wire#w1
      JumpCoil( End_G7 )
   END_RUNG
   // the same network as SCL:
   #_w1 := #Waiting_sw_req AND #MABS.Switch_right AND NOT #Edge4;   // rising edge of #MABS.Switch_right
   #Edge4 := #MABS.Switch_right;
   #_w2 := #_w1 AND NOT #MABS.Right_Pos_reach;
   IF #_w2 THEN
       #Waiting_sw_req := FALSE;
       #Switching_right := TRUE;
       GOTO End_G7;
   END_IF;
END_REGION

REGION Network 12: Swich right -> Wait
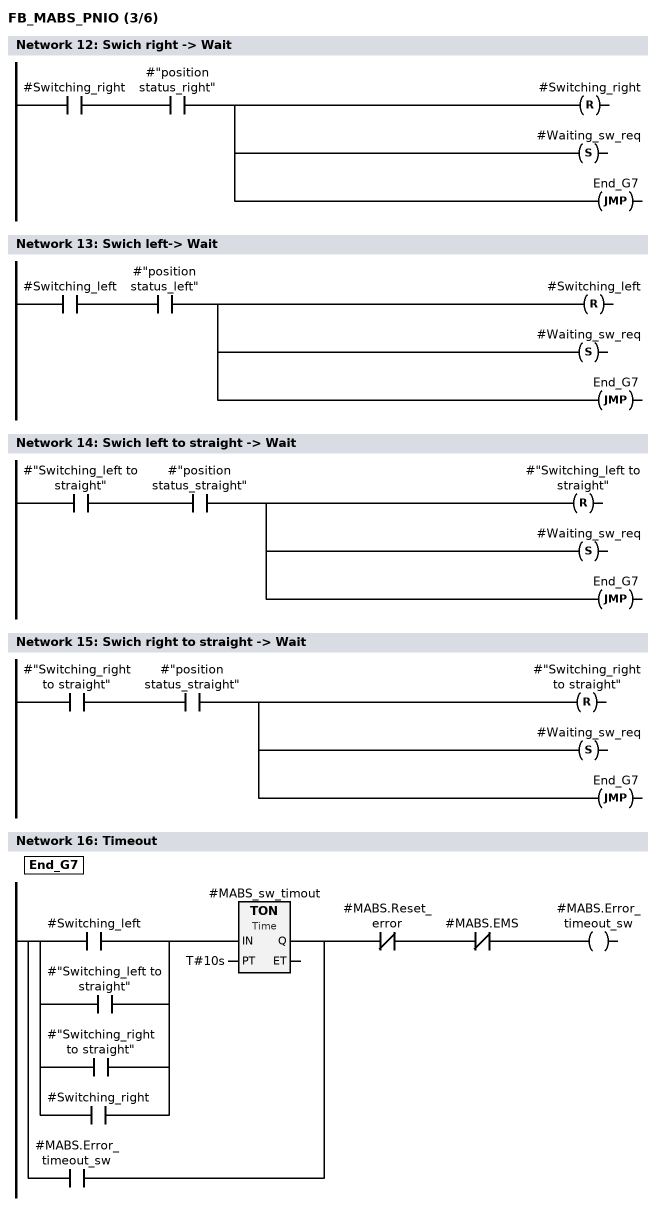
   RUNG wire#powerrail
      Contact( #Switching_right )
      Contact( #"position status_right" )
      wire#w1
      R_Coil( #Switching_right )
   END_RUNG
   RUNG wire#w1
      S_Coil( #Waiting_sw_req )
   END_RUNG
   RUNG wire#w1
      JumpCoil( End_G7 )
   END_RUNG
   // the same network as SCL:
   #_w1 := #Switching_right AND #"position status_right";
   IF #_w1 THEN
       #Switching_right := FALSE;
       #Waiting_sw_req := TRUE;
       GOTO End_G7;
   END_IF;
END_REGION

REGION Network 13: Swich left-> Wait
   RUNG wire#powerrail
      Contact( #Switching_left )
      Contact( #"position status_left" )
      wire#w1
      R_Coil( #Switching_left )
   END_RUNG
   RUNG wire#w1
      S_Coil( #Waiting_sw_req )
   END_RUNG
   RUNG wire#w1
      JumpCoil( End_G7 )
   END_RUNG
   // the same network as SCL:
   #_w1 := #Switching_left AND #"position status_left";
   IF #_w1 THEN
       #Switching_left := FALSE;
       #Waiting_sw_req := TRUE;
       GOTO End_G7;
   END_IF;
END_REGION

REGION Network 14: Swich left to straight -> Wait
   RUNG wire#powerrail
      Contact( #"Switching_left to straight" )
      Contact( #"position status_straight" )
      wire#w1
      R_Coil( #"Switching_left to straight" )
   END_RUNG
   RUNG wire#w1
      S_Coil( #Waiting_sw_req )
   END_RUNG
   RUNG wire#w1
      JumpCoil( End_G7 )
   END_RUNG
   // the same network as SCL:
   #_w1 := #"Switching_left to straight" AND #"position status_straight";
   IF #_w1 THEN
       #"Switching_left to straight" := FALSE;
       #Waiting_sw_req := TRUE;
       GOTO End_G7;
   END_IF;
END_REGION

REGION Network 15: Swich right to straight -> Wait
   RUNG wire#powerrail
      Contact( #"Switching_right to straight" )
      Contact( #"position status_straight" )
      wire#w1
      R_Coil( #"Switching_right to straight" )
   END_RUNG
   RUNG wire#w1
      S_Coil( #Waiting_sw_req )
   END_RUNG
   RUNG wire#w1
      JumpCoil( End_G7 )
   END_RUNG
   // the same network as SCL:
   #_w1 := #"Switching_right to straight" AND #"position status_straight";
   IF #_w1 THEN
       #"Switching_right to straight" := FALSE;
       #Waiting_sw_req := TRUE;
       GOTO End_G7;
   END_IF;
END_REGION

REGION Network 16: Timeout
   Label( End_G7 )
   RUNG wire#powerrail
      Contact( #Switching_left )
      wire#w1
      { S7_Templates := "time_type := Time" } #MABS_sw_timout.TON(pt := T#10s, et =>)
      wire#w2
      I_Contact( #MABS.Reset_error )
      I_Contact( #MABS.EMS )
      Coil( #MABS.Error_timeout_sw )
   END_RUNG
   RUNG wire#powerrail
      Contact( #"Switching_left to straight" )
   END_RUNG wire#w1
   RUNG wire#powerrail
      Contact( #"Switching_right to straight" )
   END_RUNG wire#w1
   RUNG wire#powerrail
      Contact( #Switching_right )
   END_RUNG wire#w1
   RUNG wire#powerrail
      Contact( #MABS.Error_timeout_sw )
   END_RUNG wire#w2
   // the same network as SCL:
   End_G7:
   #MABS_sw_timout(IN := #Switching_left OR #"Switching_left to straight" OR #"Switching_right to straight" OR #Switching_right,   // TON
                   PT := T#10s);
   #MABS.Error_timeout_sw := (#MABS_sw_timout.Q OR #MABS.Error_timeout_sw) AND NOT #MABS.Reset_error AND NOT #MABS.EMS;
END_REGION

REGION Network 17: Postion reached + origin sensor
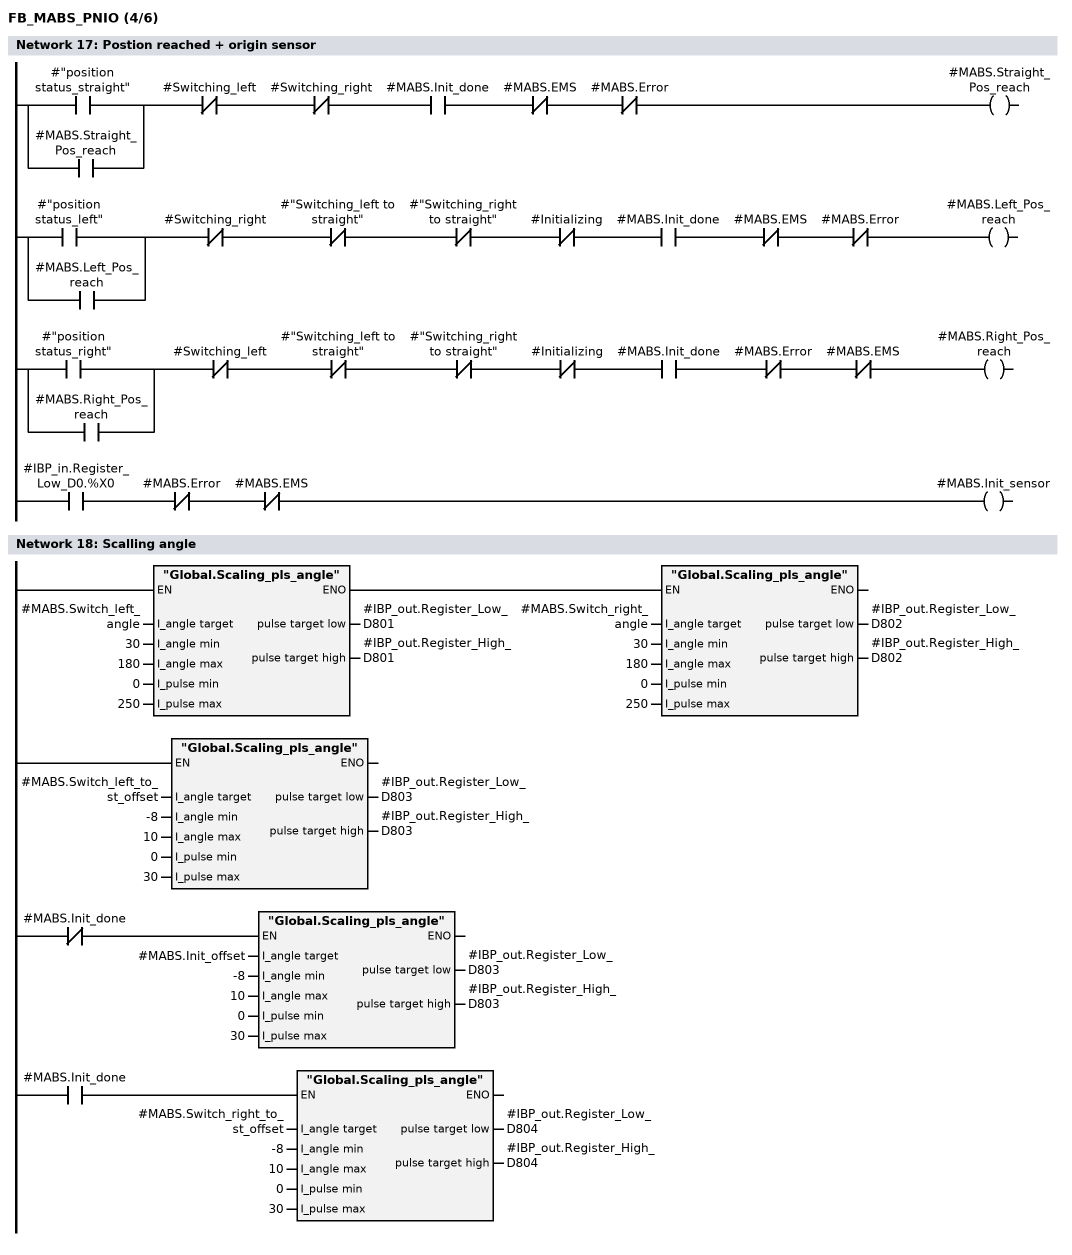
   RUNG wire#powerrail
      Contact( #"position status_straight" )
      wire#w1
      I_Contact( #Switching_left )
      I_Contact( #Switching_right )
      Contact( #MABS.Init_done )
      I_Contact( #MABS.EMS )
      I_Contact( #MABS.Error )
      Coil( #MABS.Straight_Pos_reach )
   END_RUNG
   RUNG wire#powerrail
      Contact( #MABS.Straight_Pos_reach )
   END_RUNG wire#w1
   RUNG wire#powerrail
      Contact( #"position status_left" )
      wire#w2
      I_Contact( #Switching_right )
      I_Contact( #"Switching_left to straight" )
      I_Contact( #"Switching_right to straight" )
      I_Contact( #Initializing )
      Contact( #MABS.Init_done )
      I_Contact( #MABS.EMS )
      I_Contact( #MABS.Error )
      Coil( #MABS.Left_Pos_reach )
   END_RUNG
   RUNG wire#powerrail
      Contact( #MABS.Left_Pos_reach )
   END_RUNG wire#w2
   RUNG wire#powerrail
      Contact( #"position status_right" )
      wire#w3
      I_Contact( #Switching_left )
      I_Contact( #"Switching_left to straight" )
      I_Contact( #"Switching_right to straight" )
      I_Contact( #Initializing )
      Contact( #MABS.Init_done )
      I_Contact( #MABS.Error )
      I_Contact( #MABS.EMS )
      Coil( #MABS.Right_Pos_reach )
   END_RUNG
   RUNG wire#powerrail
      Contact( #MABS.Right_Pos_reach )
   END_RUNG wire#w3
   RUNG wire#powerrail
      Contact( #IBP_in.Register_Low_D0.%X0 )
      I_Contact( #MABS.Error )
      I_Contact( #MABS.EMS )
      Coil( #MABS.Init_sensor )
   END_RUNG
   // the same network as SCL:
   #MABS.Straight_Pos_reach := (#"position status_straight" OR #MABS.Straight_Pos_reach) AND NOT #Switching_left AND NOT #Switching_right AND #MABS.Init_done AND NOT #MABS.EMS AND NOT #MABS.Error;
   #MABS.Left_Pos_reach := (#"position status_left" OR #MABS.Left_Pos_reach) AND NOT #Switching_right AND NOT #"Switching_left to straight" AND NOT #"Switching_right to straight" AND NOT #Initializing AND #MABS.Init_done AND NOT #MABS.EMS AND NOT #MABS.Error;
   #MABS.Right_Pos_reach := (#"position status_right" OR #MABS.Right_Pos_reach) AND NOT #Switching_left AND NOT #"Switching_left to straight" AND NOT #"Switching_right to straight" AND NOT #Initializing AND #MABS.Init_done AND NOT #MABS.Error AND NOT #MABS.EMS;
   #MABS.Init_sensor := #IBP_in.Register_Low_D0.%X0 AND NOT #MABS.Error AND NOT #MABS.EMS;
END_REGION

REGION Network 18: Scalling angle
   RUNG wire#powerrail
      "Global.Scaling_pls_angle"("I_angle target" := #MABS.Switch_left_angle, "I_angle min" := 30, "I_angle max" := 180, "I_pulse min" := 0, "I_pulse max" := 250, "pulse target low" => #IBP_out.Register_Low_D801, "pulse target high" => #IBP_out.Register_High_D801)
      "Global.Scaling_pls_angle"("I_angle target" := #MABS.Switch_right_angle, "I_angle min" := 30, "I_angle max" := 180, "I_pulse min" := 0, "I_pulse max" := 250, "pulse target low" => #IBP_out.Register_Low_D802, "pulse target high" => #IBP_out.Register_High_D802)
   END_RUNG
   RUNG wire#powerrail
      "Global.Scaling_pls_angle"("I_angle target" := #MABS.Switch_left_to_st_offset, "I_angle min" := -8, "I_angle max" := 10, "I_pulse min" := 0, "I_pulse max" := 30, "pulse target low" => #IBP_out.Register_Low_D803, "pulse target high" => #IBP_out.Register_High_D803)
   END_RUNG
   RUNG wire#powerrail
      I_Contact( #MABS.Init_done )
      "Global.Scaling_pls_angle"("I_angle target" := #MABS.Init_offset, "I_angle min" := -8, "I_angle max" := 10, "I_pulse min" := 0, "I_pulse max" := 30, "pulse target low" => #IBP_out.Register_Low_D803, "pulse target high" => #IBP_out.Register_High_D803)
   END_RUNG
   RUNG wire#powerrail
      Contact( #MABS.Init_done )
      "Global.Scaling_pls_angle"("I_angle target" := #MABS.Switch_right_to_st_offset, "I_angle min" := -8, "I_angle max" := 10, "I_pulse min" := 0, "I_pulse max" := 30, "pulse target low" => #IBP_out.Register_Low_D804, "pulse target high" => #IBP_out.Register_High_D804)
   END_RUNG
   // the same network as SCL:
   "Global.Scaling_pls_angle"("I_angle target" := #MABS.Switch_left_angle,
                           "I_angle min" := 30,
                           "I_angle max" := 180,
                           "I_pulse min" := 0,
                           "I_pulse max" := 250,
                           "pulse target low" => #IBP_out.Register_Low_D801,
                           "pulse target high" => #IBP_out.Register_High_D801,
                           ENO => #_w1);
   IF #_w1 THEN
       "Global.Scaling_pls_angle"("I_angle target" := #MABS.Switch_right_angle,
                               "I_angle min" := 30,
                               "I_angle max" := 180,
                               "I_pulse min" := 0,
                               "I_pulse max" := 250,
                               "pulse target low" => #IBP_out.Register_Low_D802,
                               "pulse target high" => #IBP_out.Register_High_D802);
   END_IF;
   "Global.Scaling_pls_angle"("I_angle target" := #MABS.Switch_left_to_st_offset,
                           "I_angle min" := -8,
                           "I_angle max" := 10,
                           "I_pulse min" := 0,
                           "I_pulse max" := 30,
                           "pulse target low" => #IBP_out.Register_Low_D803,
                           "pulse target high" => #IBP_out.Register_High_D803);
   IF NOT #MABS.Init_done THEN
       "Global.Scaling_pls_angle"("I_angle target" := #MABS.Init_offset,
                               "I_angle min" := -8,
                               "I_angle max" := 10,
                               "I_pulse min" := 0,
                               "I_pulse max" := 30,
                               "pulse target low" => #IBP_out.Register_Low_D803,
                               "pulse target high" => #IBP_out.Register_High_D803);
   END_IF;
   IF #MABS.Init_done THEN
       "Global.Scaling_pls_angle"("I_angle target" := #MABS.Switch_right_to_st_offset,
                               "I_angle min" := -8,
                               "I_angle max" := 10,
                               "I_pulse min" := 0,
                               "I_pulse max" := 30,
                               "pulse target low" => #IBP_out.Register_Low_D804,
                               "pulse target high" => #IBP_out.Register_High_D804);
   END_IF;
END_REGION

REGION Network 19: Swing direction
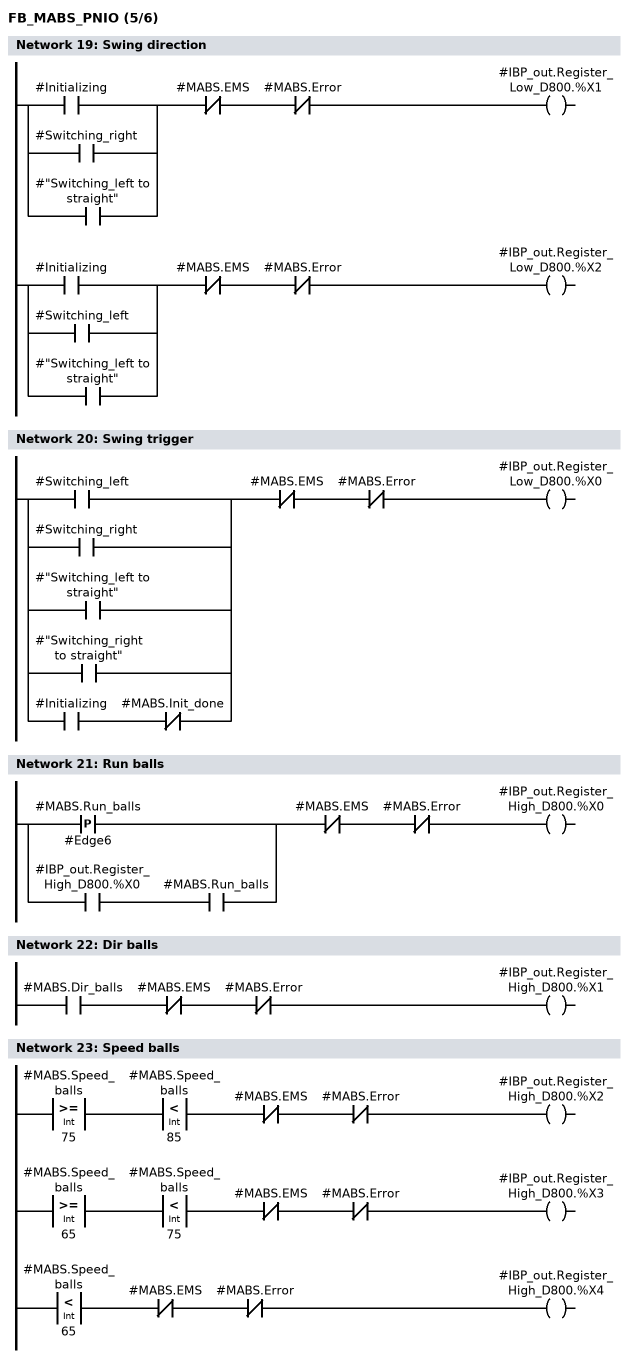
   RUNG wire#powerrail
      Contact( #Initializing )
      wire#w1
      I_Contact( #MABS.EMS )
      I_Contact( #MABS.Error )
      Coil( #IBP_out.Register_Low_D800.%X1 )
   END_RUNG
   RUNG wire#powerrail
      Contact( #Switching_right )
   END_RUNG wire#w1
   RUNG wire#powerrail
      Contact( #"Switching_left to straight" )
   END_RUNG wire#w1
   RUNG wire#powerrail
      Contact( #Initializing )
      wire#w2
      I_Contact( #MABS.EMS )
      I_Contact( #MABS.Error )
      Coil( #IBP_out.Register_Low_D800.%X2 )
   END_RUNG
   RUNG wire#powerrail
      Contact( #Switching_left )
   END_RUNG wire#w2
   RUNG wire#powerrail
      Contact( #"Switching_left to straight" )
   END_RUNG wire#w2
   // the same network as SCL:
   #IBP_out.Register_Low_D800.%X1 := (#Initializing OR #Switching_right OR #"Switching_left to straight") AND NOT #MABS.EMS AND NOT #MABS.Error;
   #IBP_out.Register_Low_D800.%X2 := (#Initializing OR #Switching_left OR #"Switching_left to straight") AND NOT #MABS.EMS AND NOT #MABS.Error;
END_REGION

REGION Network 20: Swing trigger
   RUNG wire#powerrail
      Contact( #Switching_left )
      wire#w1
      I_Contact( #MABS.EMS )
      I_Contact( #MABS.Error )
      Coil( #IBP_out.Register_Low_D800.%X0 )
   END_RUNG
   RUNG wire#powerrail
      Contact( #Switching_right )
   END_RUNG wire#w1
   RUNG wire#powerrail
      Contact( #"Switching_left to straight" )
   END_RUNG wire#w1
   RUNG wire#powerrail
      Contact( #"Switching_right to straight" )
   END_RUNG wire#w1
   RUNG wire#powerrail
      Contact( #Initializing )
      I_Contact( #MABS.Init_done )
   END_RUNG wire#w1
   // the same network as SCL:
   #IBP_out.Register_Low_D800.%X0 := (#Switching_left OR #Switching_right OR #"Switching_left to straight" OR #"Switching_right to straight" OR (#Initializing AND NOT #MABS.Init_done)) AND NOT #MABS.EMS AND NOT #MABS.Error;
END_REGION

REGION Network 21: Run balls
   RUNG wire#powerrail
      P_Contact(operand := #MABS.Run_balls, bit := #Edge6)
      wire#w1
      I_Contact( #MABS.EMS )
      I_Contact( #MABS.Error )
      Coil( #IBP_out.Register_High_D800.%X0 )
   END_RUNG
   RUNG wire#powerrail
      Contact( #IBP_out.Register_High_D800.%X0 )
      Contact( #MABS.Run_balls )
   END_RUNG wire#w1
   // the same network as SCL:
   #_w1 := #MABS.Run_balls AND NOT #Edge6;   // rising edge of #MABS.Run_balls
   #Edge6 := #MABS.Run_balls;
   #IBP_out.Register_High_D800.%X0 := (#_w1 OR (#IBP_out.Register_High_D800.%X0 AND #MABS.Run_balls)) AND NOT #MABS.EMS AND NOT #MABS.Error;
END_REGION

REGION Network 22: Dir balls
   RUNG wire#powerrail
      Contact( #MABS.Dir_balls )
      I_Contact( #MABS.EMS )
      I_Contact( #MABS.Error )
      Coil( #IBP_out.Register_High_D800.%X1 )
   END_RUNG
   // the same network as SCL:
   #IBP_out.Register_High_D800.%X1 := #MABS.Dir_balls AND NOT #MABS.EMS AND NOT #MABS.Error;
END_REGION

REGION Network 23: Speed balls
   RUNG wire#powerrail
      { S7_Templates := "SrcType := Int" } GE_Contact(in1 := #MABS.Speed_balls, in2 := 75)
      { S7_Templates := "SrcType := Int" } LT_Contact(in1 := #MABS.Speed_balls, in2 := 85)
      I_Contact( #MABS.EMS )
      I_Contact( #MABS.Error )
      Coil( #IBP_out.Register_High_D800.%X2 )
   END_RUNG
   RUNG wire#powerrail
      { S7_Templates := "SrcType := Int" } GE_Contact(in1 := #MABS.Speed_balls, in2 := 65)
      { S7_Templates := "SrcType := Int" } LT_Contact(in1 := #MABS.Speed_balls, in2 := 75)
      I_Contact( #MABS.EMS )
      I_Contact( #MABS.Error )
      Coil( #IBP_out.Register_High_D800.%X3 )
   END_RUNG
   RUNG wire#powerrail
      { S7_Templates := "SrcType := Int" } LT_Contact(in1 := #MABS.Speed_balls, in2 := 65)
      I_Contact( #MABS.EMS )
      I_Contact( #MABS.Error )
      Coil( #IBP_out.Register_High_D800.%X4 )
   END_RUNG
   // the same network as SCL:
   #IBP_out.Register_High_D800.%X2 := (#MABS.Speed_balls >= 75) AND (#MABS.Speed_balls < 85) AND NOT #MABS.EMS AND NOT #MABS.Error;
   #IBP_out.Register_High_D800.%X3 := (#MABS.Speed_balls >= 65) AND (#MABS.Speed_balls < 75) AND NOT #MABS.EMS AND NOT #MABS.Error;
   #IBP_out.Register_High_D800.%X4 := (#MABS.Speed_balls < 65) AND NOT #MABS.EMS AND NOT #MABS.Error;
END_REGION

REGION Network 24: HMI status
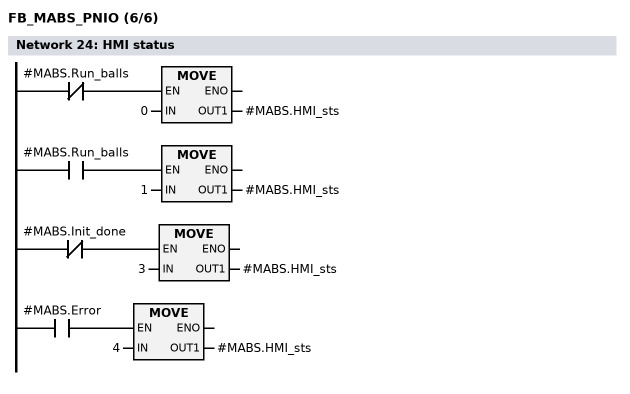
   RUNG wire#powerrail
      I_Contact( #MABS.Run_balls )
      Move(in := 0, out1 => #MABS.HMI_sts)
   END_RUNG
   RUNG wire#powerrail
      Contact( #MABS.Run_balls )
      Move(in := 1, out1 => #MABS.HMI_sts)
   END_RUNG
   RUNG wire#powerrail
      I_Contact( #MABS.Init_done )
      Move(in := 3, out1 => #MABS.HMI_sts)
   END_RUNG
   RUNG wire#powerrail
      Contact( #MABS.Error )
      Move(in := 4, out1 => #MABS.HMI_sts)
   END_RUNG
   // the same network as SCL:
   IF NOT #MABS.Run_balls THEN #MABS.HMI_sts := 0; END_IF;
   IF #MABS.Run_balls THEN #MABS.HMI_sts := 1; END_IF;
   IF NOT #MABS.Init_done THEN #MABS.HMI_sts := 3; END_IF;
   IF #MABS.Error THEN #MABS.HMI_sts := 4; END_IF;
END_REGION
END_FUNCTION_BLOCK

FUNCTION "Scaling_pls_angle" : Void   // FC12, LAD
// stored: Namespace Global, SetENOAutomatically false
   VAR_INPUT
      "I_angle target" : Int;
      "I_angle min" : Int;
      "I_angle max" : Int;
      "I_pulse min" : Int;
      "I_pulse max" : Int;
   END_VAR
   VAR_OUTPUT
      "pulse target low" : Byte;
      "pulse target high" : Byte;
   END_VAR
   VAR_TEMP
      R_pulse_calcul : Real;
      R_angle_calcul : Real;
      pulse_target_int : Int;
      Int4 : Int;
      Int5 : Int;
      Real1 : Real;
      Real2 : Real;
      Real3 : Real;
      Real4 : Real;
   END_VAR
BEGIN

REGION Network 1: Convert diff in real
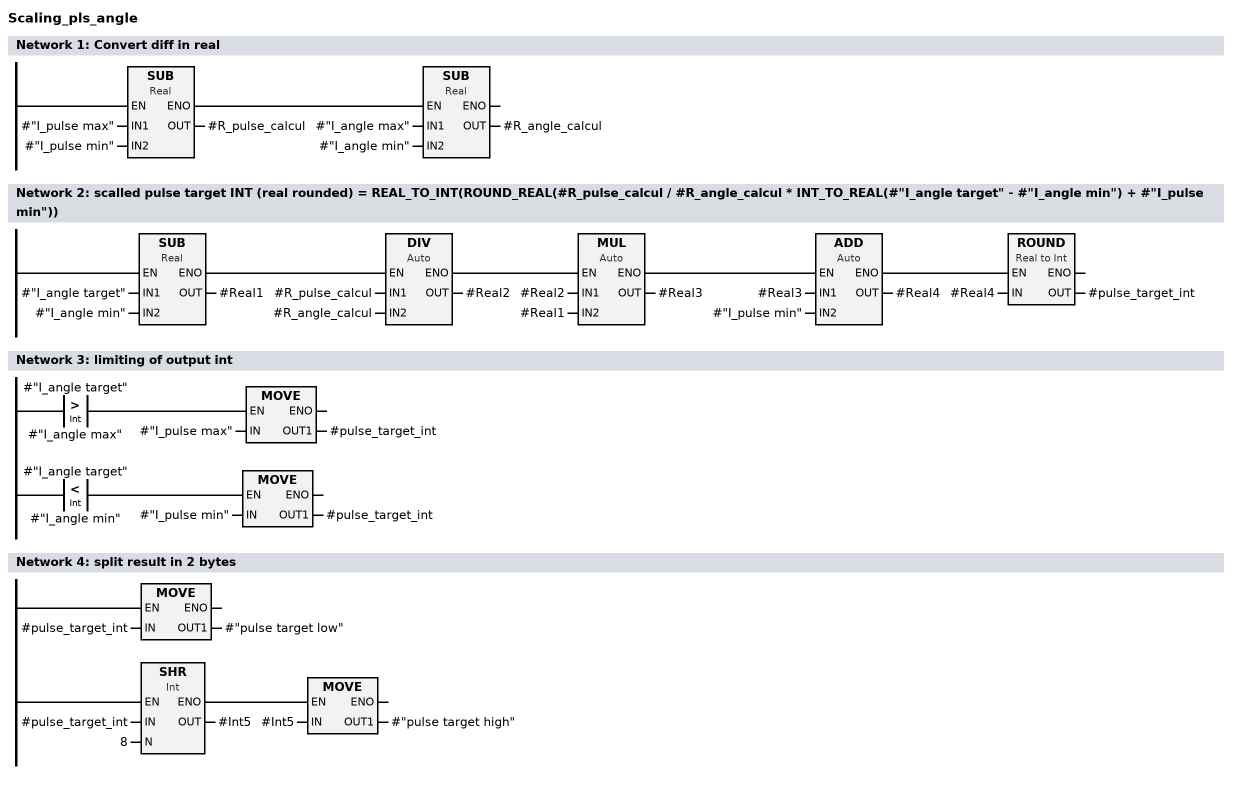
   RUNG wire#powerrail
      { S7_Templates := "SrcType := Real" } Sub(in1 := #"I_pulse max", in2 := #"I_pulse min", out => #R_pulse_calcul)
      { S7_Templates := "SrcType := Real" } Sub(in1 := #"I_angle max", in2 := #"I_angle min", out => #R_angle_calcul)
   END_RUNG
   // the same network as SCL:
   #R_pulse_calcul := #"I_pulse max" - #"I_pulse min";
   #R_angle_calcul := #"I_angle max" - #"I_angle min";
END_REGION

REGION Network 2: scalled pulse target INT (real rounded) = REAL_TO_INT(ROUND_REAL(#R_pulse_calcul / #R_angle_calcul * INT_TO_REAL(#"I_angle target" - #"I_angle min") + #"I_pulse min"))
   RUNG wire#powerrail
      { S7_Templates := "SrcType := Real" } Sub(in1 := #"I_angle target", in2 := #"I_angle min", out => #Real1)
      Div(in1 := #R_pulse_calcul, in2 := #R_angle_calcul, out => #Real2)
      Mul(in1 := #Real2, in2 := #Real1, out => #Real3)
      Add(in1 := #Real3, in2 := #"I_pulse min", out => #Real4)
      { S7_Templates := "[SrcType := Real, DestType := Int]" } Round(in := #Real4, out => #pulse_target_int)
   END_RUNG
   // the same network as SCL:
   #Real1 := #"I_angle target" - #"I_angle min";
   #Real2 := #R_pulse_calcul / #R_angle_calcul;
   #Real3 := #Real2 * #Real1;
   #Real4 := #Real3 + #"I_pulse min";
   #pulse_target_int := ROUND(#Real4);
END_REGION

REGION Network 3: limiting of output int
   RUNG wire#powerrail
      { S7_Templates := "SrcType := Int" } GT_Contact(in1 := #"I_angle target", in2 := #"I_angle max")
      Move(in := #"I_pulse max", out1 => #pulse_target_int)
   END_RUNG
   RUNG wire#powerrail
      { S7_Templates := "SrcType := Int" } LT_Contact(in1 := #"I_angle target", in2 := #"I_angle min")
      Move(in := #"I_pulse min", out1 => #pulse_target_int)
   END_RUNG
   // the same network as SCL:
   IF #"I_angle target" > #"I_angle max" THEN #pulse_target_int := #"I_pulse max"; END_IF;
   IF #"I_angle target" < #"I_angle min" THEN #pulse_target_int := #"I_pulse min"; END_IF;
END_REGION

REGION Network 4: split result in 2 bytes
   RUNG wire#powerrail
      Move(in := #pulse_target_int, out1 => #"pulse target low")
   END_RUNG
   RUNG wire#powerrail
      { S7_Templates := "SrcType := Int" } Shr(in := #pulse_target_int, n := 8, out => #Int5)
      Move(in := #Int5, out1 => #"pulse target high")
   END_RUNG
   // the same network as SCL:
   #"pulse target low" := #pulse_target_int;
   #Int5 := SHR(IN := #pulse_target_int, N := 8);
   #"pulse target high" := #Int5;
END_REGION
END_FUNCTION

FUNCTION "FC_SafetyStandard" : Void
{ S7_Optimized_Access := 'TRUE' ; Published := 'TRUE' }
VERSION : 0.1

BEGIN
	// ==========================================================================================================================================
	// Company        : LogTech, s.r.o.
	// Created by     : Mahmoud Elnady
	// Block          : FC_SafetyStandard
	// Project        : Lékárna Chrudim
	// Project number : 23-157
	// ==========================================================================================================================================
	
	REGION safety to standard: - without delay
	    
	    // All zone estop status
	    "DB_SafetyStandard".ToStandard.EstopActive :=
	    
	    NOT "FSIDB_Main_Safety_RTG1".Pair1.Q OR 
	    NOT "FSIDB_Main_Safety_RTG1".Pair2.Q OR
	    NOT "FSIDB_Main_Safety_RTG1".Pair3.Q OR
	    NOT "FSIDB_Main_Safety_RTG1".Pair4.Q OR
	    NOT "FSIDB_Main_Safety_RTG1".Pair5.Q OR
	    NOT "FSIDB_Main_Safety_RTG1".Pair6.Q OR
	    NOT "FSIDB_Main_Safety_RTG1".Pair7.Q OR
	    NOT "FSIDB_Main_Safety_RTG1".Pair8.Q OR
	    NOT "FSIDB_Main_Safety_RTG1".Pair9.Q OR
	    NOT "FSIDB_Main_Safety_RTG1".Pair10.Q;
	    
	END_REGION
	
	REGION Press Reset
	    
	    // reset needed / Ack. Req. 
	    // can be reseted when zone estop status is active and zone estop is released
	    
	    "DB_SafetyStandard".PressReset :=
	    "FSIDB_Main_Safety_RTG1".Pair1.ACK_REQ OR
	    "FSIDB_Main_Safety_RTG1".Pair2.ACK_REQ OR
	    "FSIDB_Main_Safety_RTG1".Pair3.ACK_REQ OR
	    "FSIDB_Main_Safety_RTG1".Pair4.ACK_REQ OR
	    "FSIDB_Main_Safety_RTG1".Pair5.ACK_REQ OR
	    "FSIDB_Main_Safety_RTG1".Pair6.ACK_REQ OR
	    "FSIDB_Main_Safety_RTG1".Pair7.ACK_REQ OR
	    "FSIDB_Main_Safety_RTG1".Pair8.ACK_REQ OR
	    "FSIDB_Main_Safety_RTG1".Pair9.ACK_REQ OR
	    "FSIDB_Main_Safety_RTG1".Pair10.ACK_REQ;
	    
	END_REGION
	
	REGION Hold alarm Off
	    
	    // hold alarm message OFF
	    IF "DB_SafetyStandard".ToStandard.EstopActive
	    THEN
	        "DB_SafetyStandard".holdAlarmOff := TRUE;
	    END_IF;
	    
	    // release hold after preset time
	    
	    "DB_SafetyStandard".holdAlarmOffTimer(IN := NOT "DB_SafetyStandard".ToStandard.EstopActive,
	                                          PT := t#15s);
	    
	    IF "DB_SafetyStandard".holdAlarmOffTimer.Q THEN
	        "DB_SafetyStandard".holdAlarmOff := FALSE;
	    END_IF;
	    
	END_REGION
	
	REGION to HMI
	    //Main
	    "DB_SafetyStandard".ToHMI."EstopPB -MCC001+MCC001-SF1" := NOT "MCC001+MCC001-SF1";
	    //"DB_SafetyStandard".ToHMI."PhaseOK -MCC001" := NOT "PhaseOK -MCC100";
	    //Zone 1
	    "DB_SafetyStandard".ToHMI."EstopPB -ZONA1+A1.1.1-SF1" := NOT "ZONA1+A1.1.1-SF1";
	    "DB_SafetyStandard".ToHMI."EstopPB -ZONA1+A1.1.10-SF1" := NOT "ZONA1+A1.1.10-SF1";
	    "DB_SafetyStandard".ToHMI."EstopPB -ZONA1+A1.2.1-SF1" := NOT "ZONA1+A1.2.1-SF1";
	    "DB_SafetyStandard".ToHMI."EstopPB -ZONA1+B1.22.1-SF1" := NOT "ZONA1+B1.22.1-SF1";
	    "DB_SafetyStandard".ToHMI."EstopPB -ZONA1+C1.3.1-SF1" := NOT "ZONA1+C1.3.1-SF1";
	    "DB_SafetyStandard".ToHMI."EstopPB -ZONA1+B1.12.1-SF1" := NOT "ZONA1+B1.12.1-SF1";
	    "DB_SafetyStandard".ToHMI."EstopPB -ZONA1+B1.15.1-SF1" := NOT "ZONA1+B1.15.1-SF1";
	    "DB_SafetyStandard".ToHMI."EstopPB -ZONA1+B1.17.3-SF1" := NOT "ZONA1+B1.17.3-SF1";
	    //Zone 2
	    "DB_SafetyStandard".ToHMI."EstopPB -ZONA2+D1.11.1-SF1" := NOT "ZONA2+D1.11.1-SF1";
	    "DB_SafetyStandard".ToHMI."EstopPB -ZONA2+E1.1.2-SF1" := NOT "ZONA2+E1.1.2-SF1";
	    "DB_SafetyStandard".ToHMI."EstopPB -ZONA2+A1.10.3-SF1" := NOT "ZONA2+A1.10.3-SF1";
	    "DB_SafetyStandard".ToHMI."EstopPB -ZONA2+A1.12.1-SF1" := NOT "ZONA2+A1.12.1-SF1";
	    "DB_SafetyStandard".ToHMI."EstopPB -ZONA2+A1.16.8-SF1" := NOT "ZONA2+A1.16.8-SF1";
	    "DB_SafetyStandard".ToHMI."EstopPB -ZONA2+B1.17.0-SF1" := NOT "ZONA2+B1.17.0-SF1";
	    "DB_SafetyStandard".ToHMI."EstopPB -ZONA2+A2.4.5-SF1" := NOT "ZONA2+A2.4.5-SF1";
	    "DB_SafetyStandard".ToHMI."EstopPB -ZONA2+G1.5.3-SF1" := NOT "ZONA2+G1.5.3-SF1";
	    "DB_SafetyStandard".ToHMI."EstopPB -ZONA2+G1.7.1-SF1" := NOT "ZONA2+G1.7.1-SF1";
	    
	END_REGION
	
	
	
	
	
END_FUNCTION

NAMESPACE EmptyLine
FUNCTION_BLOCK FB_EmptyLine
{ S7_Optimized_Access := 'TRUE' ; Published := 'TRUE' }
VERSION : 0.1
   VAR 
      "J1.1.1" { S7_SetPoint := 'False'} : _.Global.FB_Conveyor;
      "J1.1.2" : _.Global.FB_Conveyor;
      "J1.1.3" : _.Global.FB_Conveyor;
      "J1.1.4" : _.Global.FB_Conveyor;
      "J1.1.5" : _.Global.FB_Conveyor;
      "J1.1.6" : _.Global.FB_Conveyor;
      "J1.1.7" : _.Global.FB_Conveyor;
      "J1.1.8" : _.Global.FB_Conveyor;
      "J1.1.9" : _.Global.FB_Conveyor;
      "J1.1.10" : _.Global.FB_Conveyor;
      "J1.1.11" : _.Global.FB_Conveyor;
      "J1.1.12" : _.Global.FB_Conveyor;
      "J1.1.13" : _.Global.FB_Conveyor;
      "J1.1.14" : _.Global.FB_Conveyor;
      "J1.1.15" : _.Global.FB_Conveyor;
      "J1.1.16" : _.Global.FB_Conveyor;
      "J1.2.1" : _.Global.FB_Conveyor;
      "J1.2.2" : _.Global.FB_Conveyor;
      "J1.2.3" : _.Global.FB_Conveyor;
      "J2.1.1" : _.Global.FB_Conveyor;
      "J2.1.2" : _.Global.FB_Conveyor;
      "J2.1.3" : _.Global.FB_Conveyor;
      "J2.1.4" : _.Global.FB_Conveyor;
      "J2.1.5" : _.Global.FB_Conveyor;
      "J2.1.6" : _.Global.FB_Conveyor;
      "J2.1.7" : _.Global.FB_Conveyor;
      "J2.1.8" : _.Global.FB_Conveyor;
      "J2.1.9" : _.Global.FB_Conveyor;
      "J2.1.10" : _.Global.FB_Conveyor;
      "J2.1.11" : _.Global.FB_Conveyor;
      "J2.1.12" : _.Global.FB_Conveyor;
      "J2.1.13" : _.Global.FB_Conveyor;
      "J2.1.14" : _.Global.FB_Conveyor;
      "J2.1.15" : _.Global.FB_Conveyor;
      "J2.2.1" : _.Global.FB_Conveyor;
      "J2.2.2" : _.Global.FB_Conveyor;
      "J2.3.1" : _.Global.FB_Conveyor;
      "J2.4.1" : _.Global.FB_Conveyor;
      "J1.2.4" : _.Global.FB_Conveyor;
      "J1.2.5" : _.Global.FB_Conveyor;
      "J1.3.1" : _.Global.FB_Conveyor;
      "J1.3.2" : _.Global.FB_Conveyor;
      "J1.4.1" : _.Global.FB_Conveyor;
      "J1.4.2" : _.Global.FB_Conveyor;
      "J1.4.3" : _.Global.FB_Conveyor;
      "J1.4.4" : _.Global.FB_Conveyor;
      "J1.4.5" : _.Global.FB_Conveyor;
      "J1.4.6" : _.Global.FB_Conveyor;
      "J1.4.7" : _.Global.FB_Conveyor;
      "J1.5.1" : _.Global.FB_Conveyor;
      "J1.5.2" : _.Global.FB_Conveyor;
      "J1.5.3" : _.Global.FB_Conveyor;
      "J1.5.4" : _.Global.FB_Conveyor;
      "J1.6.1" : _.Global.FB_MABS;
      "J1.6.2" : _.Global.FB_MABS;
      "J1.7.1" : _.Global.FB_Conveyor;
      "J1.7.2" : _.Global.FB_Conveyor;
      "J1.8.1" : _.Global.FB_Conveyor;
      "J1.8.2" : _.Global.FB_Conveyor;
      "J1.9.1" : _.Global.FB_Conveyor;
      "J1.10.1" : _.Global.FB_Conveyor;
      "J1.11.1" : _.Global.FB_Conveyor;
      "J1.11.2" : _.Global.FB_Conveyor;
      "J1.11.3" : _.Global.FB_Conveyor;
      "J1.11.4" : _.Global.FB_Conveyor;
      "J1.11.5" : _.Global.FB_Conveyor;
      "J1.11.6" : _.Global.FB_Conveyor;
      "J1.11.7" : _.Global.FB_Conveyor;
      "J1.11.8" : _.Global.FB_Conveyor;
      "J1.11.9" : _.Global.FB_Conveyor;
      "J1.11.10" : _.Global.FB_Conveyor;
      "J1.11.11" : _.Global.FB_Conveyor;
      "J1.11.12" : _.Global.FB_Conveyor;
      "J1.11.13" : _.Global.FB_Conveyor;
      "K1.1.1" : _.Global.FB_Conveyor;
      "K1.2.1" : _.Global.FB_Conveyor;
      "K1.3.1" : _.Global.FB_Conveyor;
      "K1.4.1" : _.Global.FB_Conveyor;
      "K1.4.2" : _.Global.FB_Conveyor;
      "K1.4.3" : _.Global.FB_Conveyor;
      "K1.4.4" : _.Global.FB_Conveyor;
      "K1.4.5" : _.Global.FB_Conveyor;
      "K1.4.6" : _.Global.FB_Conveyor;
      "K1.4.7" : _.Global.FB_Conveyor;
      "K1.4.8" : _.Global.FB_Conveyor;
      "K1.4.9" : _.Global.FB_Conveyor;
      "K1.4.10" : _.Global.FB_Conveyor;
      "K1.5.1" : _.Global.FB_Conveyor;
      "K1.5.2" : _.Global.FB_Conveyor;
      "K1.5.3" : _.Global.FB_Conveyor;
      "K1.5.4" : _.Global.FB_Conveyor;
      "K1.5.5" : _.Global.FB_Conveyor;
      "K1.5.6" : _.Global.FB_Conveyor;
      "K1.5.7" : _.Global.FB_Conveyor;
      "K1.5.8" : _.Global.FB_Conveyor;
      "K1.6.1" : _.Global.FB_Conveyor;
      "K1.6.2" : _.Global.FB_Conveyor;
      "K1.7.1" : _.Global.FB_Conveyor;
      "K1.7.2" : _.Global.FB_Conveyor;
      "K1.8.1" : _.Global.FB_Conveyor;
      "K1.8.2" : _.Global.FB_Conveyor;
      "K1.8.3" : _.Global.FB_Conveyor;
      "K1.9.1" : _.Global.FB_Conveyor;
      "K1.9.2" : _.Global.FB_Conveyor;
      "K1.9.3" : _.Global.FB_Conveyor;
      "K1.9.4" : _.Global.FB_Conveyor;
      "K1.9.5" : _.Global.FB_Conveyor;
      "K1.9.6" : _.Global.FB_Conveyor;
      "K1.9.7" : _.Global.FB_Conveyor;
      "K1.10.1" : _.Global.FB_Conveyor;
   END_VAR


BEGIN
	// ==========================================================================================================================================
	// Company        : LogTech, s.r.o.
	// Created by     : Anton Vinoth Soundraraj
	// Block          : FB_LineB1
	// Project        : Lékarna DC Chrudim
	// Project number : 23-157
	// ==========================================================================================================================================
	
	REGION J1.1.1
	    //J1.1.1
	    #"J1.1.1"(ConveyorID:=_."J1.1.1",
	              ConveyorSensor:=_."ASiGW-MCC001-bw143-C1: Input"."Sensor J1.1.1",
	                   Fault:= DB_UDI.EmptyLine.Fault.Stop.Conveyor[_."J1.1.1"],
	                   Upstream:= DB_UDI.EmptyLine.Upstream.Conveyor[_."J1.1.1"],
	                   Downstream:= DB_UDI.EmptyLine.DownstreamAcu.Stop.Conveyor[_."J1.1.1"],
	                   Interlock:= DB_UDI.EmptyLine.Interlock.Stop.Conveyor[_."J1.1.1"],
	                   RunForward=>_."ASiGW-MCC001-bw143-C1: Output"."Motor J1.1.1",
	                   WriteAsiDir=>_."ASiGW-MCC001-bw143-C1: Output"."Dir J1.1.1");
	
	END_REGION
	
	REGION J1.1.2
	    //J1.1.2
	    #"J1.1.2"(ConveyorID:=_."J1.1.2",
	              ConveyorSensor:=_."ASiGW-MCC001-bw143-C1: Input"."Sensor J1.1.2",
	                   Fault:= DB_UDI.EmptyLine.Fault.Stop.Conveyor[_."J1.1.2"],
	                   Upstream:= DB_UDI.EmptyLine.Upstream.Conveyor[_."J1.1.2"],
	                   Downstream:= DB_UDI.EmptyLine.DownstreamAcu.Stop.Conveyor[_."J1.1.2"],
	                   Interlock:= DB_UDI.EmptyLine.Interlock.Stop.Conveyor[_."J1.1.2"],
	                   RunForward=>_."ASiGW-MCC001-bw143-C1: Output"."Motor J1.1.2",
	                   WriteAsiDir=>_."ASiGW-MCC001-bw143-C1: Output"."Dir J1.1.2");
	
	END_REGION
	
	REGION J1.1.3
	    //J1.1.3
	    #"J1.1.3"(ConveyorID:=_."J1.1.3",
	              ConveyorSensor:=_."ASiGW-MCC001-bw143-C1: Input"."Sensor J1.1.11",
	                   Fault:= DB_UDI.EmptyLine.Fault.Stop.Conveyor[_."J1.1.3"],
	                   Upstream:= DB_UDI.EmptyLine.Upstream.Conveyor[_."J1.1.3"],
	                   Downstream:= DB_UDI.EmptyLine.DownstreamAcu.Stop.Conveyor[_."J1.1.3"],
	                   Interlock:= DB_UDI.EmptyLine.Interlock.Stop.Conveyor[_."J1.1.3"],
	                   RunForward=>_."ASiGW-MCC001-bw143-C1: Output"."Motor J1.1.3",
	                   WriteAsiDir=>_."ASiGW-MCC001-bw143-C1: Output"."Dir J1.1.3");
	     END_REGION
	
	REGION J1.1.4
	    //J1.1.4
	    #"J1.1.4"(ConveyorID:=_."J1.1.4",
	              ConveyorSensor:=_."ASiGW-MCC001-bw143-C1: Input"."Sensor J1.1.11",
	                   Fault:= DB_UDI.EmptyLine.Fault.Stop.Conveyor[_."J1.1.4"],
	                   Upstream:= DB_UDI.EmptyLine.Upstream.Conveyor[_."J1.1.4"],
	                   Downstream:= DB_UDI.EmptyLine.DownstreamAcu.Stop.Conveyor[_."J1.1.4"],
	                   Interlock:= DB_UDI.EmptyLine.Interlock.Stop.Conveyor[_."J1.1.4"],
	                   RunForward=>_."ASiGW-MCC001-bw143-C1: Output"."Motor J1.1.4",
	                   WriteAsiDir=>_."ASiGW-MCC001-bw143-C1: Output"."Dir J1.1.4");
	
	END_REGION
	
